VAR_GLOBAL  (* GVL_META_GOVERNANCE_FABRIC *)
  Meta_Governance_Valid : BOOL := FALSE;
  Meta_Governance_Granted : BOOL := FALSE;
  Meta_Governance_Quarantine_Active : BOOL := TRUE;
  Governance_Graph_Acyclic : BOOL := FALSE;
  Authority_Rooting_Valid : BOOL := FALSE;
  Independent_Validation_Preserved : BOOL := FALSE;
  Meta_Consistency_Coherent : BOOL := FALSE;
  Recursive_Trust_Boundaries_Stable : BOOL := FALSE;
  Validator_Independence_Valid : BOOL := FALSE;
  CrossLayer_Causality_Grounded : BOOL := FALSE;
  Bootstrap_Validation_Absent : BOOL := FALSE;
  SelfReference_Elimination_Valid : BOOL := FALSE;
  Recursive_Authority_Dependency_Detected : BOOL := FALSE;
  Circular_Validation_Chain_Detected : BOOL := FALSE;
  SelfJustifying_Governance_State_Detected : BOOL := FALSE;
  Epistemic_Recursion_Leakage_Detected : BOOL := FALSE;
  Authority_Bootstrap_Paradox_Detected : BOOL := FALSE;
  Meta_Consistency_Erosion_Detected : BOOL := FALSE;
  Meta_Governance_Epoch : UDINT := 0;
  Meta_Governance_Epoch_Coherent : BOOL := FALSE;
  Meta_Governance_Last_Update_MS : UDINT := 0;
  Meta_Governance_Lease_Expired : BOOL := TRUE;
  Meta_Governance_Last_Error_Code : UDINT := 0;
  Meta_Governance_Last_Error_Text : STRING(160) := '';
  Meta_Governance_Invalidation_Count : UDINT := 0;
END_VAR

VAR_GLOBAL  (* GVL_RECOVERY_REACTIVATION_CONTROL_FABRIC *)
  Recovery_Reactivation_Control_Valid : BOOL := FALSE;
  Recovery_Reactivation_Control_Granted : BOOL := FALSE;
  Recovery_Reactivation_Boundary_Stable : BOOL := FALSE;
  CrossSubsystem_Reactivation_Consistent : BOOL := FALSE;
  Reactivation_Energy_Boundary_Safe : BOOL := FALSE;
  Reactivation_Causality_Grounded : BOOL := FALSE;
  Reactivation_Ordering_Stable : BOOL := FALSE;
  Unsafe_Reactivation_Ordering_Detected : BOOL := FALSE;
  Partial_Reactivation_Leak_Detected : BOOL := FALSE;
  CrossSubsystem_Reactivation_Fork : BOOL := FALSE;
  Recovery_Reactivation_Epoch : UDINT := 0;
END_VAR

VAR_GLOBAL  (* GVL_GLOBAL_AUTHORITY_SYNC *)
  Global_Authority_Sync_Valid : BOOL := FALSE;
  Global_Authority_Sync_Granted : BOOL := FALSE;
  Global_Authority_Sync_Quarantine_Active : BOOL := TRUE;
  Heating_Authority_Coherent : BOOL := FALSE;
  Ventilation_Authority_Coherent : BOOL := FALSE;
  Water_Authority_Coherent : BOOL := FALSE;
  Access_Authority_Coherent : BOOL := FALSE;
  Lighting_Authority_Coherent : BOOL := FALSE;
  Cross_Domain_Epoch_Coherent : BOOL := FALSE;
  Distributed_Authority_Generation_Coherent : BOOL := FALSE;
  Global_Causality_Timeline_Stable : BOOL := FALSE;
  Multi_Domain_Recovery_Coherent : BOOL := FALSE;
  Authority_Epoch_Fragmentation_Detected : BOOL := FALSE;
  Partial_Recovery_SplitBrain_Detected : BOOL := FALSE;
  Cross_Domain_Replay_Skew_Detected : BOOL := FALSE;
  Distributed_Authority_Divergence_Detected : BOOL := FALSE;
  Global_Causality_Desynchronization_Detected : BOOL := FALSE;
  Multi_Domain_Chronology_Drift_Detected : BOOL := FALSE;
  Global_Authority_Epoch : UDINT := 0;
  Global_Authority_Epoch_Coherent : BOOL := FALSE;
  Global_Authority_Last_Update_MS : UDINT := 0;
  Global_Authority_Lease_Expired : BOOL := TRUE;
  Global_Authority_Last_Error_Code : UDINT := 0;
  Global_Authority_Last_Error_Text : STRING(160) := '';
  Global_Authority_Invalidation_Count : UDINT := 0;
END_VAR

{attribute 'qualified_only'}
VAR_GLOBAL  (* GVL_SAFETY_RECOVERY_CONFIG *)
  G_Stabilization_Delay_MS : UDINT := 5000;
  G_Stable_Time_Required_MS : UDINT := 3000;
  G_Cooldown_Time_MS : UDINT := 10000;
END_VAR

VAR_GLOBAL  (* GVL_DISTRIBUTED_FORWARD_PROGRESS_FABRIC *)
  Distributed_Forward_Progress_Valid : BOOL := FALSE;
  Distributed_Forward_Progress_Granted : BOOL := FALSE;
  Distributed_Forward_Progress_Canonical : BOOL := FALSE;
  Cluster_Progress_Consensus_Stable : BOOL := FALSE;
  Distributed_Recovery_Progress_Valid : BOOL := FALSE;
  Distributed_Progress_Causality_Valid : BOOL := FALSE;
  Cluster_Execution_Lineage_Coherent : BOOL := FALSE;
  Distributed_Livelock_Detected : BOOL := FALSE;
  Cluster_Progress_Fork_Detected : BOOL := FALSE;
  Distributed_Consensus_Progress_Deadlock : BOOL := FALSE;
  Distributed_Forward_Progress_Epoch : UDINT := 0;
END_VAR

VAR_GLOBAL  (* GVL_TELEMETRY *)
  Telemetry_Runtime_Valid : BOOL := FALSE;
  Telemetry_Freshness_Valid : BOOL := FALSE;
  Telemetry_Lease_Expired : BOOL := TRUE;
  Telemetry_Quarantine_Active : BOOL := TRUE;
  Command_Telemetry_Causality_Valid : BOOL := FALSE;
  Command_Telemetry_Divergence_Detected : BOOL := TRUE;
  Command_Epoch : UDINT := 0;
  Telemetry_Epoch : UDINT := 0;
  Last_Acknowledged_Command_Epoch : UDINT := 0;
  Actuator_Feedback_Valid : BOOL := FALSE;
  Actuator_Feedback_Fresh : BOOL := FALSE;
  Physical_Effect_Confirmed : BOOL := FALSE;
  Physical_Effect_Finalized : BOOL := FALSE;
  Physical_Target_Converged : BOOL := FALSE;
  Physical_Stable_Window_OK : BOOL := FALSE;
  Physical_Oscillation_Detected : BOOL := FALSE;
  Physical_Transition_Active : BOOL := FALSE;
  Physical_Convergence_Replay_Suspected : BOOL := FALSE;
  Telemetry_Replay_Suspected : BOOL := FALSE;
  Last_Physical_Ack_Time_MS : UDINT := 0;
  Last_Physical_Convergence_MS : UDINT := 0;
  Telemetry_Last_Error_Code : UDINT := 0;
  Telemetry_Last_Error_Text : STRING(160) := '';
  Telemetry_Invalidation_Count : UDINT := 0;
END_VAR

VAR_GLOBAL RETAIN  (* GVL_PERSISTENT *)
  P_System_Mode : E_System_Operating_Mode;
  P_Safety_Gas_Latched : BOOL;
  P_Safety_Smoke_Latched : BOOL;
  P_Safety_Leak_Latched : BOOL;
  P_DHW_Heating_Active : BOOL;
  P_Valid : BOOL;
END_VAR

VAR_GLOBAL  (* GVL_WATER_OUTPUT *)
  DO_Water_Valve_35_Close : BOOL := FALSE;
  DO_Water_Valve_36_Close : BOOL := FALSE;
  DO_Water_Zone_Enable : ARRAY[1..GVL_CONSTANTS.C_MAX_WATER_ZONES] OF BOOL;
END_VAR

VAR_GLOBAL  (* GVL_PEER_SESSION *)
  Remote_Session_Valid : BOOL := FALSE;
  Remote_Last_Refresh_MS : UDINT := 0;
  Remote_Runtime_Epoch : ULINT := 0;
  Remote_Snapshot_Epoch : ULINT := 0;
  Remote_Boot_Generation : ULINT := 0;
  Remote_Fencing_Token : ULINT := 0;
  Remote_Publication_Allowed : BOOL := FALSE;
  Remote_Runtime_Healthy : BOOL := FALSE;
END_VAR

{attribute 'qualified_only'}
VAR_GLOBAL  (* GVL_TEST_PANEL *)
  G_Enable : BOOL := FALSE;
  G_Scenario_ID : INT := 1;
  G_Scenario_ID_Prev : INT := 0;
  G_Scenario_Run : BOOL := FALSE;
  G_Scenario_Active : BOOL := FALSE;
  G_UI_00_Header : STRING(200) := '=== TEST PANEL ===';
  G_UI_01_Test : STRING(200) := 'Select G_Scenario_ID';
  G_UI_02_Change : STRING(200) := 'CHANGE: set scenario inputs';
  G_UI_03_Expected : STRING(200) := 'EXPECTED: see scenario instruction';
  G_UI_04_Result : STRING(200) := 'RESULT: Idle';
  G_UI_05_Error : STRING(200) := 'ERROR: -';
  G_UI_06_Actual : STRING(200) := 'ACTUAL: see numeric fields below';
  G_UI_07_Separator : STRING(200) := '----------------------------------------';
  G_UI_10_Numeric_Block : STRING(200) := 'NUMERIC: Base / Expected / Actual / Delta';
  G_UI_11_Array_Block : STRING(200) := 'ARRAYS: Manifold expected / actual / enabled';
  G_UI_12_State_Block : STRING(200) := 'STATE: Safety / Block / Budget / Preheat';
  G_Run_Counter : UDINT := 0;
  G_Last_Scenario_ID : INT := 0;
  G_Last_Result_Passed : BOOL := TRUE;
  G_Last_Fail_Code : UDINT := 0;
  G_Reset_Results_Request : BOOL := FALSE;
  G_Reset_Inputs_Request : BOOL := FALSE;
  G_Current_Test_Name : STRING(200) := '';
  G_Expected_Summary : STRING(200) := '';
  G_Actual_Summary : STRING(200) := '';
  G_Test_Result_Line : STRING(200) := 'Idle';
  G_Last_Result_Line : STRING(200) := '';
  G_Error_Text : STRING(200) := '';
  G_System_State_Line : STRING(200) := '';
  G_Selected_Circuit : INT := 1;
  G_Input_Policy_Bias : INT := 0;
  G_Input_Guest_Preheat_Request : BOOL := FALSE;
  G_Input_Guest_Preheat_Enabled : BOOL := TRUE;
  G_Input_Guest_Preheat_Boost : INT := 2;
  G_Input_Max_Thermal_Budget : REAL := 2.0;
  G_Input_Block_Heating : BOOL := FALSE;
  G_Input_Safety_Stop : BOOL := FALSE;
  G_Input_Circuit_Enable : ARRAY[1..GVL_CONSTANTS.C_MAX_HEATING_CIRCUITS] OF BOOL;
  G_Input_Circuit_Bias : ARRAY[1..GVL_CONSTANTS.C_MAX_HEATING_CIRCUITS] OF INT;
  G_Input_Circuit_Guest_Preheat : ARRAY[1..GVL_CONSTANTS.C_MAX_HEATING_CIRCUITS] OF BOOL;
  G_Test_Description : STRING(200) := 'Idle';
  G_Test_What_To_Change : STRING(200) := '';
  G_Test_Expected_Text : STRING(200) := '';
  G_Result_Mapped_Manifold : INT := 0;
  G_Result_Base_Priority : INT := 0;
  G_Result_Expected_Adjusted_Priority : INT := 0;
  G_Result_Actual_Adjusted_Priority : INT := 0;
  G_Result_Delta : INT := 0;
  G_Result_Manifold_Base_Priority : ARRAY[1..GVL_CONSTANTS.C_MAX_MANIFOLDS] OF INT;
  G_Result_Manifold_Expected_Priority : ARRAY[1..GVL_CONSTANTS.C_MAX_MANIFOLDS] OF INT;
  G_Result_Manifold_Actual_Priority : ARRAY[1..GVL_CONSTANTS.C_MAX_MANIFOLDS] OF INT;
  G_Result_Manifold_Delta : ARRAY[1..GVL_CONSTANTS.C_MAX_MANIFOLDS] OF INT;
  G_Result_Manifold_Allowed : ARRAY[1..GVL_CONSTANTS.C_MAX_MANIFOLDS] OF BOOL;
  G_Result_Manifold_Enabled : ARRAY[1..GVL_CONSTANTS.C_MAX_MANIFOLDS] OF BOOL;
  G_Result_Used_Thermal_Budget : REAL := 0.0;
  G_Result_Budget_Exceeded : BOOL := FALSE;
  G_Result_Passed : BOOL := TRUE;
  G_Result_Status_Msg : STRING(200) := 'Idle';
  G_Result_Fail_Code : UDINT := 0;
END_VAR

VAR_GLOBAL  (* GVL_LIGHTING_OUTPUT *)
  AO_Lighting_Levels : ARRAY[1..GVL_CONSTANTS.C_MAX_LIGHT_ZONES] OF UINT;
  AO_Blinds_Positions : ARRAY[1..GVL_CONSTANTS.C_MAX_BLINDS] OF UINT;
  DO_Sockets : ARRAY[1..GVL_CONSTANTS.C_MAX_SOCKETS] OF BOOL;
END_VAR

VAR_GLOBAL  (* GVL_DETERMINISTIC_RECOVERY_PATH_FABRIC *)
  Deterministic_Recovery_Path_Valid : BOOL := FALSE;
  Deterministic_Recovery_Path_Granted : BOOL := FALSE;
  Deterministic_Recovery_Path_Quarantine_Active : BOOL := TRUE;
  Deterministic_Recovery_Path_Canonical : BOOL := FALSE;
  Recovery_Lineage_Causality_Valid : BOOL := FALSE;
  Recovery_Physical_Convergence_Stable : BOOL := FALSE;
  Recovery_Timeline_Monotonic : BOOL := FALSE;
  Recovery_Causality_Grounded : BOOL := FALSE;
  Recovery_Path_Continuity_Valid : BOOL := FALSE;
  Distributed_Recovery_Consensus_Valid : BOOL := FALSE;
  Unsafe_Recovery_Path_Detected : BOOL := FALSE;
  Recovery_Path_Divergence_Detected : BOOL := FALSE;
  Recovery_Causality_Break_Detected : BOOL := FALSE;
  Distributed_Recovery_Fork_Detected : BOOL := FALSE;
  Deterministic_Recovery_Path_Epoch : UDINT := 0;
  Deterministic_Recovery_Path_Last_Update_MS : UDINT := 0;
END_VAR

VAR_GLOBAL  (* GVL_ENERGY_CAUSALITY_FABRIC *)
  Energy_Causality_Valid : BOOL := FALSE;
  Energy_Causality_Granted : BOOL := FALSE;
  Energy_Causality_Quarantine_Active : BOOL := TRUE;
  Hydraulic_Energy_State_Valid : BOOL := FALSE;
  Thermal_Energy_State_Valid : BOOL := FALSE;
  Electrical_Load_State_Valid : BOOL := FALSE;
  Motor_Energy_Envelope_Valid : BOOL := FALSE;
  Distributed_Load_Coherent : BOOL := FALSE;
  Energy_Envelope_Stable : BOOL := FALSE;
  Transient_Load_Stable : BOOL := FALSE;
  Thermal_Accumulation_Stable : BOOL := FALSE;
  Recovery_Energy_Coherent : BOOL := FALSE;
  DryRun_Energy_State_Detected : BOOL := FALSE;
  Thermal_Extraction_Divergence_Detected : BOOL := FALSE;
  Load_Synchronization_Spike_Detected : BOOL := FALSE;
  Hydraulic_Energy_Starvation_Detected : BOOL := FALSE;
  Distributed_Transient_Overload_Detected : BOOL := FALSE;
  Energy_Recovery_Instability_Detected : BOOL := FALSE;
  Energy_Causality_Epoch : UDINT := 0;
  Energy_Causality_Epoch_Coherent : BOOL := FALSE;
  Energy_Causality_Last_Update_MS : UDINT := 0;
  Energy_Causality_Lease_Expired : BOOL := TRUE;
  Energy_Causality_Last_Error_Code : UDINT := 0;
  Energy_Causality_Last_Error_Text : STRING(160) := '';
  Energy_Causality_Invalidation_Count : UDINT := 0;
END_VAR

{attribute 'qualified_only'}
VAR_GLOBAL  (* GVL_MODBUS_SYSCOM_TRANSPORT *)
  G_Transport_Enabled : BOOL := FALSE;
  G_Transport_Attached : BOOL := FALSE;
  G_Backend_State : E_Modbus_SysCom_Backend_State := MB_SYSCOM_CLOSED;
  G_Backend_Last_Error_MS : UDINT := 0;
  G_Backend_Reconnect_Delay_MS : UDINT := 3000;
  G_Backend_Reconnect_Attempts : UDINT := 0;
  G_Backend_Online : BOOL := FALSE;
  G_TX_Request : BOOL := FALSE;
  G_TX_Buffer : ARRAY[0..255] OF BYTE;
  G_TX_Length : UINT := 0;
  G_TX_Done : BOOL := FALSE;
  G_TX_Error : BOOL := FALSE;
  G_TX_Error_Code : WORD := 0;
  G_RX_Ready : BOOL := FALSE;
  G_RX_Buffer : ARRAY[0..255] OF BYTE;
  G_RX_Length : UINT := 0;
  G_RX_Error : BOOL := FALSE;
  G_RX_Error_Code : WORD := 0;
  G_RX_State : E_Modbus_RTU_RX_State := MB_RTU_RX_IDLE;
  G_RX_Assembler_Active : BOOL := FALSE;
  G_RX_Assembler_Length : UINT := 0;
  G_RX_Assembler_Last_Byte_MS : UDINT := 0;
  G_RX_Assembler_InterFrame_MS : UDINT := 20;
  G_RX_Assembler_Overflow : BOOL := FALSE;
  G_RX_Assembler_CRC_OK : BOOL := FALSE;
  G_RX_Assembler_CRC_Frame : WORD := 0;
  G_RX_Assembler_CRC_Calc : WORD := 0;
  G_Last_TX_Request_MS : UDINT := 0;
  G_Last_TX_Done_MS : UDINT := 0;
  G_Last_RX_MS : UDINT := 0;
  G_TX_Watchdog_Timeout : BOOL := FALSE;
  G_RX_Watchdog_Timeout : BOOL := FALSE;
  G_Bus_Silent : BOOL := FALSE;
  G_Total_TX : UDINT := 0;
  G_Total_RX : UDINT := 0;
  G_Total_Errors : UDINT := 0;
  G_Total_RX_Overflow : UDINT := 0;
  G_Total_RX_Short_Frame : UDINT := 0;
  G_Total_RX_CRC_Error : UDINT := 0;
  G_Total_Reconnects : UDINT := 0;
  G_Total_TX_Watchdog : UDINT := 0;
  G_Total_RX_Watchdog : UDINT := 0;
END_VAR

VAR_GLOBAL  (* GVL_PLC_FENCING *)
  PLC_Ownership_Epoch : ULINT := 0;
  PLC_Fencing_Token : ULINT := 0;
  PLC_Ownership_Valid : BOOL := FALSE;
  PLC_Semantic_Authority_Valid : BOOL := FALSE;
  PLC_Heartbeat_Only_Mode : BOOL := FALSE;
  PLC_Lease_Active : BOOL := FALSE;
  PLC_Lease_Expired : BOOL := FALSE;
  PLC_Lease_Timeout_MS : UDINT := 5000;
  PLC_Last_Lease_Refresh_MS : UDINT := 0;
  PLC_Last_Authority_Validation_MS : UDINT := 0;
  PLC_Split_Brain_Detected : BOOL := FALSE;
  PLC_Stale_Owner_Detected : BOOL := FALSE;
  PLC_Asymmetric_Partition_Detected : BOOL := FALSE;
  PLC_Forced_Safe_Quarantine : BOOL := FALSE;
  PLC_Last_Error_Code : UDINT := 0;
  PLC_Last_Error_Text : STRING(160) := '';
  PLC_Fencing_Invalidation_Count : UDINT := 0;
END_VAR

VAR_GLOBAL  (* GVL_AUTHORITY_REVOCATION *)
  Authority_Revocation_Active : BOOL := FALSE;
  Authority_Revocation_Propagated : BOOL := FALSE;
  Authority_Fail_Closed_Valid : BOOL := FALSE;
  Snapshot_Authority_Revoked : BOOL := FALSE;
  Sensor_Consensus_Authority_Revoked : BOOL := FALSE;
  Telemetry_Causality_Authority_Revoked : BOOL := FALSE;
  Physical_Authority_Epoch_Revoked : BOOL := FALSE;
  Authority_Lineage_Revoked : BOOL := FALSE;
  PreOutput_Authority_Revoked : BOOL := FALSE;
  Physical_IO_Release_Denied : BOOL := FALSE;
  Quarantine_Fabric_Active : BOOL := FALSE;
  Revocation_Order_Valid : BOOL := FALSE;
  Revocation_Replay_Suspected : BOOL := FALSE;
  Partial_Revocation_Detected : BOOL := FALSE;
  Stale_Downstream_Authority_Detected : BOOL := FALSE;
  Revocation_Epoch : UDINT := 0;
  Revocation_Last_Update_MS : UDINT := 0;
  Revocation_Last_Error_Code : UDINT := 0;
  Revocation_Last_Error_Text : STRING(160) := '';
  Revocation_Invalidation_Count : UDINT := 0;
END_VAR

VAR_GLOBAL  (* GVL_PROVENANCE_CONTINUITY_FABRIC *)
  Provenance_Continuity_Valid : BOOL := FALSE;
  Provenance_Continuity_Granted : BOOL := FALSE;
  Provenance_Continuity_Quarantine_Active : BOOL := TRUE;
  Recovery_Provenance_Reattested : BOOL := FALSE;
  Authority_Resurrection_Authentic : BOOL := FALSE;
  Federation_Rejoin_Provenance_Valid : BOOL := FALSE;
  PostRecovery_TrustSeed_Coherent : BOOL := FALSE;
  CrossEpoch_Provenance_Continuity_Stable : BOOL := FALSE;
  Recovery_Epoch_Authenticity_Valid : BOOL := FALSE;
  Distributed_Rejoin_Attestation_Coherent : BOOL := FALSE;
  Authority_Restoration_Provenance_Grounded : BOOL := FALSE;
  Provenance_Lease_Continuity_Valid : BOOL := FALSE;
  Stale_Provenance_Resurrection_Detected : BOOL := FALSE;
  Recovered_Authority_Without_Reattestation_Detected : BOOL := FALSE;
  Federation_Rejoin_Without_Provenance_Detected : BOOL := FALSE;
  CrossEpoch_Trust_Continuity_Broken : BOOL := FALSE;
  Recovery_Trust_Seed_Drift_Detected : BOOL := FALSE;
  Provenance_Resurrection_Bypass_Detected : BOOL := FALSE;
  Provenance_Continuity_Epoch : UDINT := 0;
  Provenance_Continuity_Epoch_Coherent : BOOL := FALSE;
  Provenance_Continuity_Last_Update_MS : UDINT := 0;
  Provenance_Continuity_Lease_Expired : BOOL := TRUE;
  Provenance_Continuity_Last_Error_Code : UDINT := 0;
  Provenance_Continuity_Last_Error_Text : STRING(160) := '';
  Provenance_Continuity_Invalidation_Count : UDINT := 0;
END_VAR

{attribute 'qualified_only'}
VAR_GLOBAL  (* GVL_COMMAND *)
  G_Gas_Valve_Close : BOOL := FALSE;
  G_Boiler_Stop : BOOL := FALSE;
  G_Supply_100_Req : BOOL := FALSE;
  G_Supply_80_Req : BOOL := FALSE;
  G_Vent_PV3_Boost : BOOL := FALSE;
  G_Exhaust_100_Req : BOOL := FALSE;
  G_Vent_Stop : BOOL := FALSE;
  G_Close_Valve_35 : BOOL := FALSE;
  G_Close_Valve_36 : BOOL := FALSE;
  G_Gate_Open : BOOL;
  G_Wicket_Open : BOOL;
  G_Lock_1_Open : BOOL;
  G_Lock_1_Close : BOOL;
  G_Lock_2_Open : BOOL;
  G_Lock_2_Close : BOOL;
  G_Reset_Errors : BOOL := FALSE;
  G_Scenario_Request : E_SCENARIO_TYPE := E_SCENARIO_TYPE.SCENARIO_NONE;
  G_Scenario_Request_Operator : E_SCENARIO_TYPE := E_SCENARIO_TYPE.SCENARIO_NONE;
  G_Arm_Req : BOOL;
  G_Disarm_Req : BOOL;
  G_PIN_Code : STRING(4);
  G_RFID_Tag : STRING(20);
  G_2FA_Code_In : STRING(6);
  G_Send_2FA_Req : BOOL;
  G_2FA_Code_Out : STRING(6);
  G_Lighting_Override : ARRAY[1..GVL_CONSTANTS.C_MAX_LIGHT_ZONES] OF BYTE;
  G_Blinds_Override : ARRAY[1..GVL_CONSTANTS.C_MAX_BLINDS] OF BYTE;
  G_Socket_Override : ARRAY[1..GVL_CONSTANTS.C_MAX_SOCKETS] OF BOOL;
  CMD_Set_Manifold_Pump_In_Service : ARRAY[1..GVL_CONSTANTS.C_MAX_MANIFOLDS] OF BOOL;
  CMD_Set_DHW_Heating_Pump_In_Service : BOOL;
  CMD_Set_DHW_Circ_Pump_In_Service : BOOL;
  CMD_Dangerous_Action_Confirm : BOOL;
  CMD_Dangerous_Action_Request : BOOL;
  CMD_User_Access_Level : INT := 0;
  CMD_Valve_Test_Open : BOOL;
  CMD_Valve_Test_Close : BOOL;
  CMD_Valve_Test_Confirm : BOOL;
  CMD_Water_Valve_Test_Open : BOOL;
  CMD_Water_Valve_Test_Close : BOOL;
  CMD_Water_Valve_Test_Confirm : BOOL;
  CMD_Gas_Valve_Test_Open : BOOL;
  CMD_Gas_Valve_Test_Close : BOOL;
  CMD_Gas_Valve_Test_Confirm : BOOL;
  CMD_Water_Selective_Recover : BOOL;
  CMD_Gas_Selective_Recover : BOOL;
END_VAR

{attribute 'qualified_only'}
VAR_GLOBAL  (* GVL_TEST_PANEL_RESULT *)
  G_Enable : BOOL := FALSE;
  G_Scenario_ID : INT := 0;
  G_Scenario_Run : BOOL := FALSE;
  G_Scenario_Active : BOOL := FALSE;
  G_Test_Result_Line : STRING(200) := 'Idle';
  G_Result_Passed : BOOL := FALSE;
  G_Result_Status_Msg : STRING(200) := 'Idle';
  G_Result_Fail_Code : UDINT := 0;
  G_Result_Base_Priority : INT := 0;
  G_Result_Expected_Adjusted_Priority : INT := 0;
  G_Result_Actual_Adjusted_Priority : INT := 0;
  G_Result_Delta : INT := 0;
  G_Result_Budget_Exceeded : BOOL := FALSE;
  G_Result_Used_Thermal_Budget : REAL := 0.0;
  G_Result_Manifold_Enabled : ARRAY[1..GVL_CONSTANTS.C_MAX_MANIFOLDS] OF BOOL;
END_VAR

{attribute 'qualified_only'}
VAR_GLOBAL  (* GVL_Water_Isolation_Authority *)
  G_Authority_State : ARRAY[1..GVL_CONSTANTS.C_MAX_FLOOD_SENSORS] OF ST_Water_Isolation_Authority_State;
  G_Any_Selective_Authority_Allowed : BOOL;
  G_Any_Global_Fallback_Required : BOOL;
  G_Any_Authority_Denied : BOOL;
  G_Authority_Valid : BOOL;
  G_Last_Update_MS : UDINT;
  G_Status_Code : UINT;
  G_Status_Text : STRING(128);
END_VAR

{attribute 'qualified_only'}
VAR_GLOBAL  (* GVL_HEATING_POLICY_CONFIG *)
  G_Guest_Preheat_Enabled : BOOL := TRUE;
  G_Guest_Preheat_Priority_Boost : INT := 2;
  G_Guest_Preheat_Max_Duration_MS : UDINT := 7200000;
  G_Zone_Schedule : ARRAY[1..GVL_CONSTANTS.C_MAX_ZONES, 1..3] OF ST_Heating_Schedule_Event;
END_VAR

{attribute 'qualified_only'}
VAR_GLOBAL  (* GVL_Water_Topology_Validation *)
  G_Validation_State : ARRAY[1..64] OF ST_Water_Topology_Validation_State;
  G_Any_Invalid : BOOL;
  G_Any_Ambiguous : BOOL;
  G_Any_Global_Fallback_Required : BOOL;
  G_Runtime_Valid : BOOL;
  G_Last_Update_MS : UDINT;
  G_Status_Code : UINT;
  G_Status_Text : STRING(128);
END_VAR

{attribute 'qualified_only'}
VAR_GLOBAL  (* GVL_TIME_SERVICE *)
  G_Now_MS : UDINT;
  G_Time_Of_Day_MS : UDINT;
  G_Current_TOD : TOD;
  G_Day_Of_Week : INT;
  G_Last_Now_MS : UDINT;
  G_Delta_MS : UDINT;
  G_Wrap_Detected : BOOL;
  G_Sim_Enabled : BOOL;
  G_Sim_Frozen : BOOL;
  G_Sim_Time_Scale : REAL := 1.0;
  G_Sim_Now_MS : UDINT;
  G_Sim_Time_Of_Day_MS : UDINT;
  G_Sim_Day_Of_Week : INT := 1;
END_VAR

VAR_GLOBAL  (* GVL_INTENT_SYSTEM *)
  I_Source_Valid : BOOL := FALSE;
  I_Last_Update_Cycle : UDINT := 0;
  I_Last_Update_MS : UDINT := 0;
  I_Mode_Safe_Stop_Active : BOOL := FALSE;
  I_Mode_Degraded_Active : BOOL := FALSE;
  I_Mode_Freeze_Protection_Active : BOOL := FALSE;
  I_Preheat_Request : BOOL := FALSE;
  I_Freeze_Request : BOOL := FALSE;
  I_Scenario_Request_Allowed : BOOL := FALSE;
  I_Operator_Scenario_Block : BOOL := FALSE;
  I_Gateway_Command_Valid : BOOL := FALSE;
  I_Gateway_Command_Type : INT := 0;
  I_Gateway_Writes_Allowed : BOOL := FALSE;
  I_Reset_Errors_Request : BOOL := FALSE;
  I_Config_Apply_Allowed : BOOL := FALSE;
  I_Time_Sync_Allowed : BOOL := FALSE;
  I_Temperature_Write_Allowed : BOOL := FALSE;
  I_Ventilation_Write_Allowed : BOOL := FALSE;
  I_Maintenance_Apply_Allowed : BOOL := FALSE;
  I_Lighting_Overrides_Block : BOOL := FALSE;
  I_Blinds_Overrides_Block : BOOL := FALSE;
  I_Socket_Overrides_Block : BOOL := FALSE;
  I_Access_Open_Allowed : BOOL := FALSE;
  I_Manual_Override_Allowed : BOOL := FALSE;
  I_Dangerous_Action_Allowed : BOOL := FALSE;
END_VAR

VAR_GLOBAL  (* GVL_EVENT *)
  G_Event_Log : ARRAY[0..63] OF ST_EVENT;
  G_Event_Head : UINT;
  G_Event_ID_Counter : UDINT;
END_VAR

{attribute 'qualified_only'}
VAR_GLOBAL  (* GVL_Heating_Source_Stability *)
  G_State : ARRAY[1..GVL_CONSTANTS.C_MAX_HEATING_CIRCUITS] OF ST_Heating_Runtime_Source_Instability_State;
END_VAR

VAR_GLOBAL  (* GVL_PHYSICAL_TRANSACTION *)
  Physical_Transaction_Valid : BOOL := FALSE;
  Physical_Transaction_Granted : BOOL := FALSE;
  Physical_Transaction_Quarantine_Active : BOOL := TRUE;
  Physical_Transaction_Epoch : UDINT := 0;
  Physical_Transaction_Command_Epoch : UDINT := 0;
  Physical_Transaction_ACK_Epoch : UDINT := 0;
  All_Actuators_Converged : BOOL := FALSE;
  Cross_Actuator_Epoch_Coherent : BOOL := FALSE;
  Distributed_Actuation_Coherent : BOOL := FALSE;
  Stable_Plant_State_Confirmed : BOOL := FALSE;
  Valve_Transition_Confirmed : BOOL := FALSE;
  Pump_Transition_Confirmed : BOOL := FALSE;
  Damper_Transition_Confirmed : BOOL := FALSE;
  Relay_Bank_Transition_Confirmed : BOOL := FALSE;
  Flow_Stabilization_Confirmed : BOOL := FALSE;
  Pressure_Stabilization_Confirmed : BOOL := FALSE;
  Thermal_Response_Confirmed : BOOL := FALSE;
  Electrical_Load_Stabilized : BOOL := FALSE;
  Partial_Plant_Transition_Detected : BOOL := FALSE;
  Cross_Actuator_Convergence_Skew : BOOL := FALSE;
  Pump_Valve_Ordering_Race_Detected : BOOL := FALSE;
  Distributed_Actuator_Rollback_Detected : BOOL := FALSE;
  Transaction_Timeout_Detected : BOOL := FALSE;
  Brownout_Partial_Switching_Detected : BOOL := FALSE;
  Physical_Transaction_Last_Update_MS : UDINT := 0;
  Physical_Transaction_Lease_Expired : BOOL := TRUE;
  Physical_Transaction_Last_Error_Code : UDINT := 0;
  Physical_Transaction_Last_Error_Text : STRING(160) := '';
  Physical_Transaction_Invalidation_Count : UDINT := 0;
END_VAR

{attribute 'qualified_only'}
VAR_GLOBAL  (* GVL_Water_Isolation_Intent *)
  G_Zone_Close_Requested : ARRAY[1..GVL_CONSTANTS.C_MAX_FLOOD_SENSORS] OF BOOL;
  G_Valve_Group_Close_Requested : ARRAY[1..GVL_CONSTANTS.C_MAX_FLOOD_SENSORS] OF BOOL;
  G_Global_Isolation_Requested : BOOL;
  G_Intent_Valid : BOOL;
  G_Status_Code : UINT;
  G_Status_Text : STRING(128);
END_VAR

VAR_GLOBAL  (* GVL_TEMPORAL_STABILITY *)
  Temporal_Stability_Valid : BOOL := FALSE;
  Temporal_Stability_Granted : BOOL := FALSE;
  Temporal_Stability_Quarantine_Active : BOOL := TRUE;
  Stability_Observation_Window_Active : BOOL := FALSE;
  Stability_Window_Start_MS : UDINT := 0;
  Stability_Window_Elapsed_MS : UDINT := 0;
  Stability_Window_Target_MS : UDINT := 5000;
  Post_Convergence_Stable : BOOL := FALSE;
  No_Oscillation_Detected : BOOL := FALSE;
  No_Relay_Chatter_Detected : BOOL := FALSE;
  Thermal_Slope_Stable : BOOL := FALSE;
  Pressure_Stable : BOOL := FALSE;
  Flow_Stable : BOOL := FALSE;
  Post_Convergence_Oscillation_Detected : BOOL := FALSE;
  Thermal_Inertia_Rebound_Detected : BOOL := FALSE;
  Pressure_Rebound_Detected : BOOL := FALSE;
  Relay_Chatter_Detected : BOOL := FALSE;
  Pump_Cavitation_Recovery_Detected : BOOL := FALSE;
  Delayed_Actuator_Divergence_Detected : BOOL := FALSE;
  Temporal_Stability_Epoch : UDINT := 0;
  Temporal_Stability_Epoch_Coherent : BOOL := FALSE;
  Temporal_Stability_Last_Update_MS : UDINT := 0;
  Temporal_Stability_Lease_Expired : BOOL := TRUE;
  Temporal_Stability_Last_Error_Code : UDINT := 0;
  Temporal_Stability_Last_Error_Text : STRING(160) := '';
  Temporal_Stability_Invalidation_Count : UDINT := 0;
END_VAR

{attribute 'qualified_only'}
VAR_GLOBAL  (* GVL_Water_Output_Projection *)
  G_Output_Projection_State : ARRAY[1..64] OF ST_Water_Output_Projection_State;
  G_Any_Output_Projected : BOOL;
  G_Any_Projection_Denied : BOOL;
  G_Global_Fallback_Projecting : BOOL;
  G_Runtime_Valid : BOOL;
  G_Last_Update_MS : UDINT;
  G_Status_Code : UINT;
  G_Status_Text : STRING(128);
END_VAR

VAR_GLOBAL  (* GVL_OPERATIONAL_INTELLIGENCE_FABRIC *)
  Operational_Intelligence_Active : BOOL := TRUE;
  Operational_Intelligence_ReadOnly : BOOL := TRUE;
  Operational_Intelligence_NoMutation : BOOL := TRUE;
  Dominant_Instability_Source_Available : BOOL := FALSE;
  Active_Degradation_Cause_Available : BOOL := FALSE;
  Recovery_Blocker_Observed : BOOL := FALSE;
  Governance_Pressure_Hotspot_Observed : BOOL := FALSE;
  Operational_Reasoning_Consistency_Valid : BOOL := FALSE;
  Runtime_Causal_Projection_Valid : BOOL := FALSE;
  Distributed_Operational_Context_Valid : BOOL := FALSE;
  Governance_Saturation_Observed : BOOL := FALSE;
  Governance_Complexity_Pressure_Observed : BOOL := FALSE;
  Operational_Opacity_Observed : BOOL := FALSE;
  Operational_Intelligence_Epoch : UDINT := 0;
END_VAR

{attribute 'qualified_only'}
VAR_GLOBAL  (* GVL_DIAGNOSTICS_EXT *)
  G_Health_Heating : REAL := 1.0;
  G_Health_Safety : REAL := 1.0;
  G_Health_IO : REAL := 1.0;
  G_Error_Count_Heating : UDINT := 0;
  G_Error_Count_Safety : UDINT := 0;
  G_Error_Count_IO : UDINT := 0;
  G_Last_Error_Time_Heating : UDINT := 0;
  G_Last_Error_Time_Safety : UDINT := 0;
  G_Last_Error_Time_IO : UDINT := 0;
  G_Last_Update_Time : UDINT := 0;
  G_Cycle_Expected_MS : UDINT := 250;
  G_Cycle_Warning_MS : UDINT := 375;
  G_Cycle_Critical_MS : UDINT := 500;
  G_Cycle_Last_MS : UDINT := 0;
  G_Cycle_Max_MS : UDINT := 0;
  G_Cycle_Min_MS : UDINT := 0;
  G_Cycle_Avg_MS : REAL := 0.0;
  G_Cycle_Sample_Count : UDINT := 0;
  G_Cycle_Overrun_Count : UDINT := 0;
  G_Cycle_Critical_Count : UDINT := 0;
  G_Cycle_Last_Overrun_MS : UDINT := 0;
  G_Cycle_Last_Overrun_Time_MS : UDINT := 0;
  G_Cycle_Overrun_Active : BOOL := FALSE;
  G_Cycle_Critical_Active : BOOL := FALSE;
  G_Heating_State : INT := 0;  (* 0=OK,1=DEGRADED,2=CRITICAL *)
  G_Safety_State : INT := 0;
  G_IO_State : INT := 0;
END_VAR

VAR_GLOBAL  (* GVL_SAFETY_SHUTDOWN *)
  G_Safety_Mode : E_Safety_Mode := NORMAL;
  G_Safety_Active : BOOL := FALSE;
END_VAR

VAR_GLOBAL RETAIN  (* GVL_AUTHORITY_LINEAGE *)
  Authority_Lineage_Epoch : UDINT := 0;
  Authority_Lineage_Valid : BOOL := FALSE;
  Warm_Restart_Continuity_Valid : BOOL := FALSE;
  HA_Resume_Continuity_Valid : BOOL := FALSE;
  Retained_State_Integrity_Valid : BOOL := FALSE;
  Authority_Replay_Suspected : BOOL := FALSE;
  Retained_State_Skew_Detected : BOOL := FALSE;
  Partial_Authority_Resurrection_Detected : BOOL := FALSE;
  Epoch_Lineage_Discontinuity_Detected : BOOL := FALSE;
  Last_Physical_Authority_Epoch : UDINT := 0;
  Last_Runtime_Epoch : UDINT := 0;
  Last_Output_Publication_Epoch : UDINT := 0;
  Authority_Lineage_Boot_ID : UDINT := 0;
  Authority_Lineage_Last_Update_MS : UDINT := 0;
  Authority_Lineage_Last_Error_Code : UDINT := 0;
  Authority_Lineage_Last_Error_Text : STRING(160) := '';
  Authority_Lineage_Invalidation_Count : UDINT := 0;
END_VAR

VAR_GLOBAL  (* GVL_CONTROL_TIMING_FABRIC *)
  Control_Temporal_Coherence_Valid : BOOL := FALSE;
  Control_Temporal_Coherence_Granted : BOOL := FALSE;
  Control_Temporal_Coherence_Quarantine_Active : BOOL := TRUE;
  Loop_Sampling_Coherent : BOOL := FALSE;
  Feedback_Freshness_Valid : BOOL := FALSE;
  PID_Phase_Alignment_Valid : BOOL := FALSE;
  Cross_Loop_Temporal_Stable : BOOL := FALSE;
  Multi_Rate_Causality_Coherent : BOOL := FALSE;
  Control_Snapshot_Epoch_Coherent : BOOL := FALSE;
  Feedback_Window_Stable : BOOL := FALSE;
  Loop_Execution_Phase_Stable : BOOL := FALSE;
  Temporal_Observation_Aligned : BOOL := FALSE;
  PID_Phase_Skew_Detected : BOOL := FALSE;
  Sampling_Window_Divergence_Detected : BOOL := FALSE;
  Feedback_Freshness_Aliasing_Detected : BOOL := FALSE;
  Cross_Loop_Stabilization_Lag_Detected : BOOL := FALSE;
  Multi_Rate_Oscillation_Risk_Detected : BOOL := FALSE;
  Distributed_Control_Ringing_Detected : BOOL := FALSE;
  Control_Timing_Epoch : UDINT := 0;
  Control_Timing_Epoch_Coherent : BOOL := FALSE;
  Control_Timing_Last_Update_MS : UDINT := 0;
  Control_Timing_Lease_Expired : BOOL := TRUE;
  Control_Timing_Last_Error_Code : UDINT := 0;
  Control_Timing_Last_Error_Text : STRING(160) := '';
  Control_Timing_Invalidation_Count : UDINT := 0;
END_VAR

VAR_GLOBAL  (* GVL_SEMANTIC_CONTINUITY *)
  Semantic_Continuity_Valid : BOOL := FALSE;
  Semantic_Continuity_Granted : BOOL := FALSE;
  Semantic_Continuity_Quarantine_Active : BOOL := TRUE;
  Operator_Intent_Coherent : BOOL := FALSE;
  Policy_Intent_Coherent : BOOL := FALSE;
  Adaptive_Behavior_Coherent : BOOL := FALSE;
  Recovery_Intent_Coherent : BOOL := FALSE;
  Distributed_Semantic_Coherent : BOOL := FALSE;
  Declared_System_Intent_Valid : BOOL := FALSE;
  Runtime_Goal_Alignment_Valid : BOOL := FALSE;
  Optimization_Boundary_Valid : BOOL := FALSE;
  Autonomous_Adjustment_Valid : BOOL := FALSE;
  Goal_Drift_Detected : BOOL := FALSE;
  Policy_Divergence_Detected : BOOL := FALSE;
  Adaptive_Learning_Semantic_Skew : BOOL := FALSE;
  Recovery_Intent_Mismatch_Detected : BOOL := FALSE;
  Optimization_Authority_Corruption_Detected : BOOL := FALSE;
  Distributed_Semantic_Fragmentation_Detected : BOOL := FALSE;
  Semantic_Continuity_Epoch : UDINT := 0;
  Semantic_Continuity_Epoch_Coherent : BOOL := FALSE;
  Semantic_Last_Update_MS : UDINT := 0;
  Semantic_Lease_Expired : BOOL := TRUE;
  Semantic_Last_Error_Code : UDINT := 0;
  Semantic_Last_Error_Text : STRING(160) := '';
  Semantic_Invalidation_Count : UDINT := 0;
END_VAR

VAR_GLOBAL  (* GVL_CAUSAL_NARRATIVE_FABRIC *)
  Causal_Narrative_Active : BOOL := TRUE;
  Causal_Narrative_ReadOnly : BOOL := TRUE;
  Runtime_Narrative_Available : BOOL := FALSE;
  Recovery_Narrative_Available : BOOL := FALSE;
  Authority_Narrative_Available : BOOL := FALSE;
  Temporal_Narrative_Available : BOOL := FALSE;
  Narrative_Causality_Coherent : BOOL := FALSE;
  Narrative_Runtime_Alignment_Valid : BOOL := FALSE;
  Narrative_Opacity_Observed : BOOL := FALSE;
  Narrative_Gap_Observed : BOOL := FALSE;
  Runtime_Narrative_Code : STRING(255) := '';
  Recovery_Narrative_Code : STRING(255) := '';
  Authority_Narrative_Code : STRING(255) := '';
  Causal_Narrative_Epoch : UDINT := 0;
END_VAR

VAR_GLOBAL  (* GVL_DISTRIBUTED_SAFETY_REALITY_CONSENSUS_FABRIC *)
  Distributed_Safety_Reality_Consensus_Valid : BOOL := FALSE;
  Distributed_Safety_Reality_Consensus_Granted : BOOL := FALSE;
  Distributed_Safety_Consensus_Valid : BOOL := FALSE;
  Cluster_Safety_Reality_Stable : BOOL := FALSE;
  Distributed_Observability_Reality_Equivalence : BOOL := FALSE;
  Distributed_Safety_Causality_Valid : BOOL := FALSE;
  Cluster_Safety_Lineage_Coherent : BOOL := FALSE;
  Distributed_Safety_State_Fork : BOOL := FALSE;
  Cluster_Safety_Projection_Drift : BOOL := FALSE;
  Distributed_Unsafe_State_Hidden : BOOL := FALSE;
  Distributed_Safety_Reality_Epoch : UDINT := 0;
END_VAR

{attribute 'qualified_only'}
VAR_GLOBAL  (* GVL_IO_Binding_Runtime *)
  G_Flood_Sensor_Value : ARRAY[1..64] OF BOOL;
  G_Flood_Sensor_Valid : ARRAY[1..64] OF BOOL;
  G_Water_Valve_Open_FB_Value : ARRAY[1..64] OF BOOL;
  G_Water_Valve_Open_FB_Valid : ARRAY[1..64] OF BOOL;
  G_Water_Valve_Close_FB_Value : ARRAY[1..64] OF BOOL;
  G_Water_Valve_Close_FB_Valid : ARRAY[1..64] OF BOOL;
  G_Water_Valve_Output_Channel_Valid : ARRAY[1..64] OF BOOL;
  G_Runtime_Valid : BOOL;
  G_Last_Update_MS : UDINT;
  G_Any_Invalid_Binding : BOOL;
  G_Any_Missing_Binding : BOOL;
  G_Status_Code : UINT;
  G_Status_Text : STRING(128);
END_VAR

VAR_GLOBAL  (* GVL_DISTRIBUTED_COMMIT *)
  Distributed_Commit_Epoch : ULINT := 0;
  Distributed_Commit_Reconciliation_Epoch : ULINT := 0;
  Local_Publication_Commit_Epoch : ULINT := 0;
  Peer_Publication_Commit_Epoch : ULINT := 0;
  Local_Prepare_Epoch : ULINT := 0;
  Peer_Prepare_Epoch : ULINT := 0;
  Publication_Prepare_Active : BOOL := FALSE;
  Publication_Prepare_Valid : BOOL := FALSE;
  Publication_Commit_Requested : BOOL := FALSE;
  Publication_Commit_Confirmed : BOOL := FALSE;
  Peer_Commit_Ack_Valid : BOOL := FALSE;
  Peer_Commit_Ack_Expired : BOOL := FALSE;
  Peer_Commit_Mismatch : BOOL := FALSE;
  Peer_Commit_Replay_Detected : BOOL := FALSE;
  Peer_Commit_Missing : BOOL := FALSE;
  Commit_Lease_Active : BOOL := FALSE;
  Commit_Lease_Expired : BOOL := FALSE;
  Commit_Timeout_MS : UDINT := 5000;
  Local_Commit_Last_Refresh_MS : UDINT := 0;
  Peer_Commit_Last_Refresh_MS : UDINT := 0;
  Commit_Last_Reconciliation_MS : UDINT := 0;
  Distributed_Commit_Valid : BOOL := FALSE;
  Distributed_Commit_Quarantine_Active : BOOL := FALSE;
  Distributed_Commit_Last_Error_Code : UDINT := 0;
  Distributed_Commit_Last_Error_Text : STRING(160) := '';
END_VAR

VAR_GLOBAL  (* GVL_SEMANTIC_EPOCH_INVARIANCE_FABRIC *)
  Semantic_Epoch_Invariance_Valid : BOOL := FALSE;
  Semantic_Epoch_Invariance_Granted : BOOL := FALSE;
  Semantic_Epoch_Invariance_Quarantine_Active : BOOL := TRUE;
  Authority_Semantics_Invariant : BOOL := FALSE;
  CrossEpoch_Permission_Mapping_Stable : BOOL := FALSE;
  Semantic_Intent_Continuity_Valid : BOOL := FALSE;
  Governance_Meaning_Preservation_Coherent : BOOL := FALSE;
  Semantic_Evolution_Lineage_Traceable : BOOL := FALSE;
  Explicit_Semantic_Migration_Governed : BOOL := FALSE;
  CrossEpoch_Semantic_Equivalence_Valid : BOOL := FALSE;
  Distributed_Semantic_Consensus_Stable : BOOL := FALSE;
  Semantic_Interpretation_Integrity_Valid : BOOL := FALSE;
  Semantic_Authority_Drift_Detected : BOOL := FALSE;
  CrossEpoch_Permission_Reinterpretation : BOOL := FALSE;
  Intent_To_Authority_Mismatch_Detected : BOOL := FALSE;
  Governance_Semantic_Fork_Detected : BOOL := FALSE;
  Semantic_Migration_Lineage_Gap_Detected : BOOL := FALSE;
  Distributed_Semantic_Divergence_Detected : BOOL := FALSE;
  Semantic_Epoch_Invariance_Epoch : UDINT := 0;
  Semantic_Epoch_Invariance_Epoch_Coherent : BOOL := FALSE;
  Semantic_Epoch_Invariance_Last_Update_MS : UDINT := 0;
  Semantic_Epoch_Invariance_Lease_Expired : BOOL := TRUE;
  Semantic_Epoch_Invariance_Last_Error_Code : UDINT := 0;
  Semantic_Epoch_Invariance_Last_Error_Text : STRING(160) := '';
  Semantic_Epoch_Invariance_Invalidation_Count : UDINT := 0;
END_VAR

VAR_GLOBAL  (* GVL_SAFETY_RECOVERY *)
  G_Recovery_Phase : E_Recovery_Phase := IDLE;
  G_Recovery_Active : BOOL := FALSE;
  G_Recovery_Requested : BOOL := FALSE;
  G_Recovery_Manual_Confirm : BOOL := FALSE;
  G_Recovery_Start_MS : UDINT := 0;
  G_Recovery_Stable_Since_MS : UDINT := 0;
  G_Recovery_Cooldown_Start_MS : UDINT := 0;
  G_Recovery_Exit_Allowed : BOOL := FALSE;
  G_Recovery_Abort_Reason : INT := 0;  (* 0=none, 1=safety active, 2=confidence low, 3=timeout *)
END_VAR

VAR_GLOBAL  (* GVL_HA_SESSION_REPLICATION *)
  HA_Replication_Enabled : BOOL := FALSE;
  HA_Channel_Healthy : BOOL := FALSE;
  HA_Last_TX_MS : UDINT := 0;
  HA_Last_RX_MS : UDINT := 0;
  HA_Remote_Session_Valid : BOOL := FALSE;
  HA_Remote_Last_Refresh_MS : UDINT := 0;
  HA_Remote_Runtime_Epoch : ULINT := 0;
  HA_Remote_Snapshot_Epoch : ULINT := 0;
  HA_Remote_Boot_Generation : ULINT := 0;
  HA_Remote_Fencing_Token : ULINT := 0;
  HA_Remote_Publication_Allowed : BOOL := FALSE;
  HA_Remote_Runtime_Healthy : BOOL := FALSE;
  HA_Remote_Distributed_Snapshot_Epoch : ULINT := 0;
  HA_Remote_Runtime_Snapshot_Epoch : ULINT := 0;
  HA_Remote_Publication_Epoch : ULINT := 0;
  HA_Remote_Snapshot_Immutable : BOOL := FALSE;
  HA_Remote_Snapshot_Last_Refresh_MS : UDINT := 0;
  HA_Remote_Publication_Commit_Epoch : ULINT := 0;
  HA_Remote_Prepare_Epoch : ULINT := 0;
  HA_Remote_Commit_Ack_Valid : BOOL := FALSE;
  HA_Remote_Commit_Last_Refresh_MS : UDINT := 0;
END_VAR

VAR_GLOBAL  (* GVL_EXECUTION_PROJECTION_INTEGRITY_FABRIC *)
  Execution_Projection_Integrity_Valid : BOOL := FALSE;
  Execution_Projection_Integrity_Granted : BOOL := FALSE;
  Execution_Projection_Integrity_Quarantine_Active : BOOL := TRUE;
  Execution_Authority_Projection_Consistent : BOOL := FALSE;
  CrossDomain_Actuation_Enforcement_Aligned : BOOL := FALSE;
  Physical_Execution_Governance_Canonical : BOOL := FALSE;
  Actuation_Surface_Consensus_Valid : BOOL := FALSE;
  Execution_Projection_Lineage_Coherent : BOOL := FALSE;
  Runtime_Actuation_Projection_Stable : BOOL := FALSE;
  Distributed_Execution_Equivalence_Valid : BOOL := FALSE;
  Execution_Governance_Causality_Grounded : BOOL := FALSE;
  Physical_Enforcement_Timeline_Monotonic : BOOL := FALSE;
  Execution_Projection_Divergence_Detected : BOOL := FALSE;
  Actuation_Path_Authority_Bypass_Detected : BOOL := FALSE;
  CrossDomain_Enforcement_Fork_Detected : BOOL := FALSE;
  Canonical_Governance_Execution_Lost : BOOL := FALSE;
  Runtime_Execution_Lineage_Drift_Detected : BOOL := FALSE;
  Distributed_Actuation_Reality_Fork_Detected : BOOL := FALSE;
  Execution_Projection_Integrity_Epoch : UDINT := 0;
  Execution_Projection_Integrity_Epoch_Coherent : BOOL := FALSE;
  Execution_Projection_Integrity_Last_Update_MS : UDINT := 0;
  Execution_Projection_Integrity_Lease_Expired : BOOL := TRUE;
  Execution_Projection_Integrity_Last_Error_Code : UDINT := 0;
  Execution_Projection_Integrity_Last_Error_Text : STRING(160) := '';
  Execution_Projection_Integrity_Invalidation_Count : UDINT := 0;
END_VAR

{attribute 'qualified_only'}
VAR_GLOBAL  (* GVL_Distributed_Projection_Ownership *)
  G_Projection_Ownership : ARRAY[1..128] OF ST_Distributed_Projection_Ownership;
END_VAR

VAR_GLOBAL  (* GVL_DEGRADED *)
  G_System_Degraded : BOOL := FALSE;
  G_Degraded_Mode_Active : BOOL := FALSE;
  G_Degraded_Recovery_Required : BOOL := FALSE;
END_VAR

{attribute 'qualified_only'}
VAR_GLOBAL  (* GVL_Heating_Runtime_Projection *)
  G_Circuit_Projection : ARRAY[1..GVL_CONSTANTS.C_MAX_HEATING_CIRCUITS] OF ST_Heating_Circuit_Runtime_Projection;
END_VAR

{attribute 'qualified_only'}
VAR_GLOBAL  (* GVL_SYSTEM_SIZE_CONFIG *)
  G_Active_Heating_Circuits : INT := GVL_CONSTANTS.C_MAX_HEATING_CIRCUITS;
  G_Active_Water_Zones : INT := GVL_CONSTANTS.C_MAX_WATER_ZONES;
  G_Active_Light_Zones : INT := GVL_CONSTANTS.C_MAX_LIGHT_ZONES;
  G_Active_Blinds : INT := GVL_CONSTANTS.C_MAX_BLINDS;
  G_Active_Sockets : INT := GVL_CONSTANTS.C_MAX_SOCKETS;
END_VAR

{attribute 'qualified_only'}
VAR_GLOBAL  (* GVL_CONFIG_BACKUP *)
  G_Backup_FloorHeating_Configs : ARRAY[1..GVL_CONSTANTS.C_MAX_HEATING_CIRCUITS] OF ST_FloorHeating_Circuit_Config;
  G_Backup_Max_Active_Manifolds : INT := 0;
  G_Backup_Max_Thermal_Budget : REAL := 0.0;
  G_Backup_Valid : BOOL := FALSE;
END_VAR

{attribute 'qualified_only'}
VAR_GLOBAL  (* GVL_COMMAND_POLICY_CONFIG *)
  G_PLC_Inactive_Close_Gas : BOOL := TRUE;
  G_PLC_Inactive_Stop_Boiler : BOOL := TRUE;
  G_PLC_Inactive_Block_Heating : BOOL := TRUE;
  G_PLC_Inactive_Stop_Vent : BOOL := TRUE;
  G_PLC_Inactive_Block_Water : BOOL := TRUE;
  G_Fire_Block_Heating : BOOL := TRUE;
  G_Fire_Stop_Boiler : BOOL := TRUE;
  G_Fire_Stop_Vent : BOOL := TRUE;
  G_Fire_Open_Lock_1 : BOOL := TRUE;
  G_Fire_Open_Lock_2 : BOOL := TRUE;
  G_Fire_Open_Gate : BOOL := TRUE;
  G_Fire_Open_Wicket : BOOL := TRUE;
  G_Fire_Block_Lock_Close : BOOL := TRUE;
  G_Gas_Close_Gas : BOOL := TRUE;
  G_Gas_Stop_Boiler : BOOL := TRUE;
  G_Gas_Block_Heating : BOOL := TRUE;
  G_Gas_Open_Gate : BOOL := TRUE;
  G_Gas_Open_Wicket : BOOL := TRUE;
  G_Gas_Open_Lock_1 : BOOL := FALSE;
  G_Gas_Open_Lock_2 : BOOL := FALSE;
  G_Water_Block_Water : BOOL := TRUE;
  G_GlobalStop_Block_Heating : BOOL := TRUE;
  G_GlobalStop_Stop_Boiler : BOOL := TRUE;
  G_GlobalStop_Stop_Vent : BOOL := TRUE;
  G_GlobalStop_Block_Water : BOOL := TRUE;
  G_Block_Close_When_Open_Commanded : BOOL := TRUE;
END_VAR

{attribute 'qualified_only'}
VAR_GLOBAL  (* GVL_CONFIG *)
  G_Heating_Config : ST_Heating_Config;
  G_DHW_Config : ST_DHW_Config;
  G_Security_Config : ST_Security_Global_Config;
  G_HMI_FloorHeating_Configs : ARRAY[1..GVL_CONSTANTS.C_MAX_HEATING_CIRCUITS] OF ST_FloorHeating_Circuit_Config;
  G_Heating_Circuit_To_Zone : ARRAY[1..GVL_CONSTANTS.C_MAX_HEATING_CIRCUITS] OF INT := [1, 2, 3, 4, 5, 6, 7, 8, 9, 10, 11, 12, 13, 14, 15, 16];
  G_Wet_Zone_Map : ARRAY[1..32] OF BOOL;
  G_HMI_Tariff_Settings : ST_Tariff_Config;
  G_HMI_Vent_Global_Config : ST_Ventilation_Global_Config;
  G_HMI_Scenario_Configs : ARRAY[1..GVL_CONSTANTS.C_MAX_SCENARIOS] OF ST_Scenario_Config;
  G_HMI_Flood_Config : ST_Flood_Global_Config;
  G_Flood_Global_Config : ST_Flood_Global_Config;
  G_HMI_User_Rules : ARRAY[1..GVL_CONSTANTS.C_MAX_RULES] OF ST_User_Rule;
  G_Calib_Outdoor_Temp : ST_Sensor_Calibration_Record;
  G_Calib_Supply_Temps : ARRAY[1..GVL_CONSTANTS.C_MAX_SUPPLY_TEMPS] OF ST_Sensor_Calibration_Record;
  G_Calib_Room_Temps : ARRAY[1..GVL_CONSTANTS.C_MAX_ZONES] OF ST_Sensor_Calibration_Record;
  G_Calib_Floor_Temps : ARRAY[1..GVL_CONSTANTS.C_MAX_ZONES] OF ST_Sensor_Calibration_Record;
  G_Calib_CO2 : ARRAY[1..GVL_CONSTANTS.C_MAX_ZONES] OF ST_Sensor_Calibration_Record;
  G_Calib_Humidity : ARRAY[1..GVL_CONSTANTS.C_MAX_ZONES] OF ST_Sensor_Calibration_Record;
  G_Calib_Manifold_T_Supply : ARRAY[1..GVL_CONSTANTS.C_MAX_MANIFOLDS] OF ST_Sensor_Calibration_Record;
  G_Calib_Manifold_T_Return : ARRAY[1..GVL_CONSTANTS.C_MAX_MANIFOLDS] OF ST_Sensor_Calibration_Record;
  G_Calib_Methane : ARRAY[1..GVL_CONSTANTS.C_MAX_METHANE_SENSORS] OF ST_Sensor_Calibration_Record;
  G_Calib_CO : ARRAY[1..GVL_CONSTANTS.C_MAX_CO_SENSORS] OF ST_Sensor_Calibration_Record;
  G_Valve_Test_Config : ARRAY[1..GVL_CONSTANTS.C_MAX_MANIFOLDS] OF ST_Valve_Test_Config;
  G_HMI_Apply_Settings : BOOL;
  G_HMI_Mute_Alarm : BOOL;
  G_HMI_Ack_Alarms : BOOL;
  G_HMI_Gate_Open_Req : BOOL;
  G_HMI_Wicket_Open_Req : BOOL;
  G_HMI_Lock_1_Open_Req : BOOL;
  G_HMI_Lock_1_Close_Req : BOOL;
  G_HMI_Lock_2_Open_Req : BOOL;
  G_HMI_Lock_2_Close_Req : BOOL;
  G_Access_Pulse_MS : UDINT := 500;
  G_Allowed_IPs : ARRAY[1..GVL_CONSTANTS.C_MAX_ALLOWED_IPS] OF STRING(15) := ['192.168.1.100', '192.168.1.101', '127.0.0.1', '', ''];
  G_Backup_Circulation_Pump_In_Service : BOOL := TRUE;
  G_Electric_Heater_In_Service : BOOL := TRUE;
  G_Freeze_Hardware_Retry_Count : INT := 2;
  G_Freeze_Hardware_Retry_Delay_MS : UDINT := 5000;
  G_Pump_Exercise_Enabled : BOOL := TRUE;
  G_Pump_Exercise_Interval_MS : UDINT := 604800000;
  G_Pump_Exercise_Duration_MS : UDINT := 30000;
  G_Manifold_Pump_In_Service : ARRAY[1..GVL_CONSTANTS.C_MAX_MANIFOLDS] OF BOOL := [TRUE, TRUE, TRUE, TRUE, TRUE];
  G_Manifold_Priority : ARRAY[1..GVL_CONSTANTS.C_MAX_MANIFOLDS] OF INT := [3, 3, 2, 2, 1];
  G_Manifold_Thermal_Weight : ARRAY[1..GVL_CONSTANTS.C_MAX_MANIFOLDS] OF REAL := [1.0, 1.0, 0.8, 0.8, 0.5];
  G_Max_Active_Manifolds : INT := 3;
  G_Max_Thermal_Budget : REAL := 6.0;
  G_Policy_Min_Hold_MS : UDINT := 300000;
  G_DHW_Heating_Pump_In_Service : BOOL := TRUE;
  G_DHW_Circ_Pump_In_Service : BOOL := TRUE;
  G_Water_Valve_Exercise_Enabled : BOOL := TRUE;
  G_Water_Valve_Exercise_Interval_MS : UDINT := 604800000;
  G_Water_Valve_Exercise_Duration_MS : UDINT := 15000;
  G_Water_Valve_Close_Retry_Count : INT := 2;
  G_Water_Valve_Close_Retry_Delay_MS : UDINT := 3000;
  G_OpenTherm_Enabled : BOOL := FALSE;
  G_OpenTherm_Heartbeat_Timeout_MS : UDINT := 5000;
  G_OpenTherm_Command_Ack_Timeout_MS : UDINT := 3000;
  G_OpenTherm_Register_Map : ARRAY[1..GVL_CONSTANTS.C_MAX_BOILERS] OF ST_OpenTherm_Register_Map;
  G_Modbus_RTU_Driver_Attached : BOOL := FALSE;
  G_Modbus_RTU_Port_Number : BYTE := 1;  (* 1=COM1, 2=COM2, 3=COM3, 4=COM4 *)
  G_Modbus_RTU_Baudrate : UDINT := 9600;
  G_Modbus_RTU_Parity : BYTE := 1;  (* 0=None, 1=Even, 2=Odd *)
  G_Modbus_RTU_Stop_Bits : BYTE := 1;  (* 1 or 2 *)
  G_Modbus_RTU_Data_Bits : BYTE := 8;  (* usually 8 *)
  G_Modbus_RTU_Slave_ID : BYTE := 1;
  G_Modbus_RTU_Poll_Interval_MS : UDINT := 100;
  G_Modbus_RTU_Request_Timeout_MS : UDINT := 250;
  G_Modbus_RTU_Retry_Count : INT := 2;
  G_FloorTemp_Map : ARRAY[1..GVL_CONSTANTS.C_MAX_HEATING_CIRCUITS] OF INT := [1, 2, 3, 4, 5, 6, 7, 8, 9, 10, 11, 12, 13, 14, 15, 16];
  G_RoomTemp_Map : ARRAY[1..16] OF INT := [1, 2, 3, 4, 5, 6, 7, 8, 9, 10, 11, 12, 13, 14, 15, 16];
  G_Door_Map : ARRAY[1..GVL_CONSTANTS.C_MAX_DOOR_SENSORS] OF INT := [1, 2, 3, 4, 5, 6, 7, 8];
  G_Window_Map : ARRAY[1..16] OF INT := [9, 10, 11, 12, 13, 14, 15, 16, 17, 18, 19, 20, 21, 22, 23, 24];
  C_MAX_LIGHT_ZONES : INT := 32;
  G_Evac_Exit_Zones : ARRAY[1..32] OF BOOL;
  G_Evac_Zone_Names : ARRAY[1..32] OF STRING(80);
END_VAR

{attribute 'qualified_only'}
VAR_GLOBAL  (* GVL_HMI_Config_Workflow *)
  G_Open_Editor_Request : BOOL;
  G_Validate_Request : BOOL;
  G_Activate_Request : BOOL;
  G_Rollback_Request : BOOL;
  G_Service_Mode_Active : BOOL;
  G_Operator_Ack : BOOL;
  G_Workflow_State : ST_HMI_Config_Workflow_State;
  G_Runtime_Valid : BOOL;
  G_Last_Update_MS : UDINT;
  G_Status_Code : UINT;
  G_Status_Text : STRING(160);
END_VAR

VAR_GLOBAL  (* GVL_DISTRIBUTED_EPOCH *)
  Distributed_Epoch : ULINT := 0;
  Distributed_Reconciliation_Epoch : ULINT := 0;
  Local_Runtime_Epoch : ULINT := 0;
  Peer_Runtime_Epoch : ULINT := 0;
  Local_Snapshot_Epoch : ULINT := 0;
  Peer_Snapshot_Epoch : ULINT := 0;
  Local_Boot_Generation : ULINT := 0;
  Peer_Boot_Generation : ULINT := 0;
  Local_Fencing_Token : ULINT := 0;
  Peer_Fencing_Token : ULINT := 0;
  Distributed_Epoch_Consistent : BOOL := FALSE;
  Distributed_Reconciliation_Valid : BOOL := FALSE;
  Distributed_Publication_Allowed : BOOL := FALSE;
  Peer_Lease_Active : BOOL := FALSE;
  Peer_Lease_Expired : BOOL := FALSE;
  Peer_Lease_Timeout_MS : UDINT := 5000;
  Peer_Last_Refresh_MS : UDINT := 0;
  Peer_Last_Reconciliation_MS : UDINT := 0;
  Peer_Snapshot_Stale : BOOL := FALSE;
  Peer_Runtime_Stale : BOOL := FALSE;
  Peer_Boot_Mismatch : BOOL := FALSE;
  Peer_Fencing_Conflict : BOOL := FALSE;
  Peer_Semantic_Continuity_Lost : BOOL := FALSE;
  Distributed_Quarantine_Active : BOOL := FALSE;
  Distributed_Last_Error_Code : UDINT := 0;
  Distributed_Last_Error_Text : STRING(160) := '';
END_VAR

{attribute 'qualified_only'}
VAR_GLOBAL  (* GVL_MODE *)
  G_Current_Behavior_Mode : E_Behavior_Mode := BEHAVIOR_HOME;
  G_Mode_Last_Change_TS : UDINT := 0;
  G_Mode_Code : UDINT := 0;
  G_Away_Request : BOOL := FALSE;
  G_Maintenance_Request : BOOL := FALSE;
END_VAR

VAR_GLOBAL  (* GVL_ENVIRONMENTAL_AUTHORITY *)
  Environmental_Authority_Valid : BOOL := FALSE;
  Environmental_Authority_Granted : BOOL := FALSE;
  Environmental_Quarantine_Active : BOOL := TRUE;
  External_Environment_Causally_Compatible : BOOL := FALSE;
  Utility_Environment_Stable : BOOL := FALSE;
  Hydraulic_Source_Stable : BOOL := FALSE;
  Thermal_Environment_Stable : BOOL := FALSE;
  Airflow_Environment_Stable : BOOL := FALSE;
  Mains_Quality_Valid : BOOL := FALSE;
  Supply_Water_Available : BOOL := FALSE;
  Outdoor_Airflow_Valid : BOOL := FALSE;
  Freeze_Protection_Valid : BOOL := FALSE;
  Freeze_Front_Propagation_Detected : BOOL := FALSE;
  Utility_Instability_Propagation_Detected : BOOL := FALSE;
  External_Hydraulic_Collapse_Detected : BOOL := FALSE;
  Airflow_Icing_Condition_Detected : BOOL := FALSE;
  Environmental_Rebound_Race_Detected : BOOL := FALSE;
  Environmental_Authority_Epoch : UDINT := 0;
  Environmental_Authority_Epoch_Coherent : BOOL := FALSE;
  Environmental_Last_Update_MS : UDINT := 0;
  Environmental_Lease_Expired : BOOL := TRUE;
  Environmental_Last_Error_Code : UDINT := 0;
  Environmental_Last_Error_Text : STRING(160) := '';
  Environmental_Invalidation_Count : UDINT := 0;
END_VAR

VAR_GLOBAL  (* GVL_PHYSICAL_AUTHORITY_EPOCH *)
  Physical_Authority_Epoch : UDINT := 0;
  Physical_Authority_Epoch_Valid : BOOL := FALSE;
  Snapshot_Epoch_Coherent : BOOL := FALSE;
  Consensus_Epoch_Coherent : BOOL := FALSE;
  Causality_Epoch_Coherent : BOOL := FALSE;
  PreOutput_Epoch_Coherent : BOOL := FALSE;
  Physical_Epoch_Drift_Detected : BOOL := FALSE;
  Physical_Epoch_Replay_Suspected : BOOL := FALSE;
  Partial_Epoch_Advancement_Detected : BOOL := FALSE;
  Cross_Cycle_Epoch_Skew_Detected : BOOL := FALSE;
  Physical_Authority_Lease_Expired : BOOL := TRUE;
  Physical_Authority_Quarantine_Active : BOOL := TRUE;
  Physical_Authority_Last_Update_MS : UDINT := 0;
  Physical_Authority_Last_Error_Code : UDINT := 0;
  Physical_Authority_Last_Error_Text : STRING(160) := '';
  Physical_Authority_Invalidation_Count : UDINT := 0;
END_VAR

{attribute 'qualified_only'}
VAR_GLOBAL  (* GVL_CONFIG_SIMULATION *)
  G_Simulation_Request : BOOL := FALSE;
  G_Simulation_Confirm : BOOL := FALSE;
  G_Simulation_Result_OK : BOOL := TRUE;
  G_Simulation_Error_Text : STRING(200) := '';
  G_Simulation_Last_Run_MS : UDINT := 0;
END_VAR

VAR_GLOBAL  (* GVL_RUNTIME_EPOCH *)
  Runtime_Epoch : ULINT := 0;
  Runtime_Snapshot_Valid : BOOL := FALSE;
  Runtime_Snapshot_Published : BOOL := FALSE;
  Runtime_Runtime_Barrier_OK : BOOL := TRUE;
  Runtime_Impossible_State_Detected : BOOL := FALSE;
  Runtime_Last_Validation_Time_MS : UDINT := 0;
  Runtime_Last_Error_Code : UDINT := 0;
  Runtime_Last_Error_Text : STRING(160) := '';
  Runtime_Cycle_Start_MS : UDINT := 0;
  Runtime_Cycle_End_MS : UDINT := 0;
  Runtime_PLC_Authority_Valid : BOOL := FALSE;
  Runtime_IO_Publication_Allowed : BOOL := FALSE;
  Runtime_Barrier_Block_Count : UDINT := 0;
END_VAR

{attribute 'qualified_only'}
VAR_GLOBAL RETAIN  (* GVL_Retain *)
  G_Initialized : BOOL := FALSE;  (* Флаг инициализации retain-переменных *)
  G_NVRAM_Data : ARRAY[0..12799] OF BYTE;  (* 100 * 128 = 12800 байт *)
  G_BlackBox_Buffer : ARRAY[0..GVL_CONSTANTS.C_MAX_BLACKBOX_RECORDS-1] OF ST_BlackBox_Record;
  G_BlackBox_LastIndex : INT;
  G_BlackBox_Frozen : BOOL;
  G_Presence_History : ARRAY[0..GVL_CONSTANTS.C_MAX_PRESENCE_HISTORY-1] OF WORD;  (* 168 часов * 6 записей в час = 1008 записей (битовая маска 16 ламп) *)
  G_History_Buffer : ARRAY[1..GVL_CONSTANTS.C_MAX_HISTORY_RECORDS] OF ST_History_Record;
  G_History_Write_Idx : INT := 1;
  G_History_Total_Events : UDINT;
  G_Boiler_Accumulated_MS : ARRAY[1..GVL_CONSTANTS.C_MAX_BOILERS] OF UDINT;
  G_Boiler_Work_Seconds : ARRAY[1..GVL_CONSTANTS.C_MAX_BOILERS] OF UDINT;
  G_Valve_Test_Results : ARRAY[1..GVL_CONSTANTS.C_MAX_MANIFOLDS] OF BOOL;
  G_Access_Codes : ARRAY[1..GVL_CONSTANTS.C_MAX_ACCESS_CODES] OF DWORD := [16#9BE3E0A3, 16#4A89A12D, 16#F4DBDF21, 16#90F59C65, 16#0972D346, 0, 0, 0, 0, 0];
  G_RFID_Tags : ARRAY[1..GVL_CONSTANTS.C_MAX_ACCESS_CODES] OF STRING(20) := ['A1B2C3D4', 'E5F67890', '', '', '', '', '', '', '', ''];
END_VAR

VAR_GLOBAL  (* GVL_SURVIVABILITY_INTELLIGENCE_FABRIC *)
  Survivability_Intelligence_Active : BOOL := TRUE;
  Survivability_Intelligence_ReadOnly : BOOL := TRUE;
  Survivability_Intelligence_NoActuation : BOOL := TRUE;
  Survivability_Intelligence_NoAuthorityMutation : BOOL := TRUE;
  Survivability_Intelligence_NoRecoveryMutation : BOOL := TRUE;
  System_Survivable : BOOL := FALSE;
  Degraded_But_Safe : BOOL := FALSE;
  Isolated_But_Stable : BOOL := FALSE;
  Partitioned_But_Survivable : BOOL := FALSE;
  Resource_Starved_But_Recoverable : BOOL := FALSE;
  Essential_Functions_Preserved : BOOL := FALSE;
  NonEssential_Shedding_Recommended : BOOL := FALSE;
  Telemetry_Rate_Reduction_Recommended : BOOL := FALSE;
  Heavy_Diagnostics_Defer_Recommended : BOOL := FALSE;
  Trend_Analytics_Defer_Recommended : BOOL := FALSE;
  Simulation_Defer_Recommended : BOOL := FALSE;
  LongDuration_Degradation_Observed : BOOL := FALSE;
  Chronic_Degradation_Risk_Increasing : BOOL := FALSE;
  Survivability_Pressure_Observed : BOOL := FALSE;
  Governance_Saturation_Pressure_Observed : BOOL := FALSE;
  Telemetry_Overload_Pressure_Observed : BOOL := FALSE;
  Distributed_Instability_Pressure_Observed : BOOL := FALSE;
  Survivability_Advisory_Available : BOOL := FALSE;
  Survivability_Advisory_Code : STRING(255) := '';
  Survivability_Intelligence_Epoch : UDINT := 0;
END_VAR

VAR_GLOBAL  (* GVL_OBSERVABILITY_TRUTH *)
  Observability_Truth_Valid : BOOL := FALSE;
  Observability_Truth_Granted : BOOL := FALSE;
  Observability_Truth_Quarantine_Active : BOOL := TRUE;
  HMI_Authority_Coherent : BOOL := FALSE;
  Alarm_Authority_Coherent : BOOL := FALSE;
  Trend_Authority_Coherent : BOOL := FALSE;
  Diagnostics_Authority_Coherent : BOOL := FALSE;
  History_Authority_Coherent : BOOL := FALSE;
  HMI_Epoch_Coherent : BOOL := FALSE;
  Alarm_Publication_Coherent : BOOL := FALSE;
  Trend_Causality_Coherent : BOOL := FALSE;
  Diagnostics_Causality_Coherent : BOOL := FALSE;
  Operator_Visibility_Consistent : BOOL := FALSE;
  Stale_HMI_Epoch_Detected : BOOL := FALSE;
  Alarm_Publication_Lag_Detected : BOOL := FALSE;
  Trend_Causality_Skew_Detected : BOOL := FALSE;
  Diagnostic_Truth_Race_Detected : BOOL := FALSE;
  Operator_Visibility_Fragmentation_Detected : BOOL := FALSE;
  Authority_UI_Divergence_Detected : BOOL := FALSE;
  Observability_Truth_Epoch : UDINT := 0;
  Observability_Truth_Epoch_Coherent : BOOL := FALSE;
  Observability_Last_Update_MS : UDINT := 0;
  Observability_Lease_Expired : BOOL := TRUE;
  Observability_Last_Error_Code : UDINT := 0;
  Observability_Last_Error_Text : STRING(160) := '';
  Observability_Invalidation_Count : UDINT := 0;
END_VAR

VAR_GLOBAL  (* GVL_HEATING_DIAGNOSTICS *)
  G_Manifold_Pressure_Fault : ARRAY[1..16] OF BOOL;
  G_Manifold_Current_Fault : ARRAY[1..16] OF BOOL;
  G_Manifold_Return_Temp_Fault : ARRAY[1..16] OF BOOL;
END_VAR

{attribute 'qualified_only'}
VAR_GLOBAL  (* GVL_TEST_PANEL_DEBUG *)
  G_Test_Description : STRING(200);
  G_Test_What_To_Change : STRING(200);
  G_Test_Expected_Text : STRING(200);
  G_Expected_Summary : STRING(200);
  G_Actual_Summary : STRING(200);
  G_Error_Text : STRING(200);
  G_System_State_Line : STRING(200);
  G_Input_Guest_Preheat_Request : BOOL;
  G_Input_Guest_Preheat_Enabled : BOOL;
  G_Input_Guest_Preheat_Boost : INT;
  G_Input_Max_Thermal_Budget : REAL;
  G_Input_Block_Heating : BOOL;
  G_Input_Safety_Stop : BOOL;
END_VAR

VAR_GLOBAL  (* GVL_ACCESS_OUTPUT *)
  DO_Lock_1_Open : BOOL := FALSE;
  DO_Lock_1_Close : BOOL := FALSE;
  DO_Lock_2_Open : BOOL := FALSE;
  DO_Lock_2_Close : BOOL := FALSE;
  DO_Gate_Open : BOOL := FALSE;
  DO_Wicket_Open : BOOL := FALSE;
END_VAR

VAR_GLOBAL  (* GVL_HEATING_REQUEST *)
  G_Freeze_Request : BOOL := FALSE;
  G_Target_Temperature : REAL := 0.0;
  G_Preheat_Request : BOOL := FALSE;
END_VAR

VAR_GLOBAL  (* GVL_COMPLIANCE_FEDERATION_FABRIC *)
  Compliance_Federation_Valid : BOOL := FALSE;
  Compliance_Federation_Granted : BOOL := FALSE;
  Compliance_Federation_Quarantine_Active : BOOL := TRUE;
  Regulatory_Semantics_Coherent : BOOL := FALSE;
  Certification_Boundary_Valid : BOOL := FALSE;
  Regional_Safety_Envelope_Aligned : BOOL := FALSE;
  Governance_Trust_Boundary_Stable : BOOL := FALSE;
  Policy_Compliance_Coherent : BOOL := FALSE;
  CrossJurisdiction_Authority_Aligned : BOOL := FALSE;
  Compliance_Runtime_Projection_Stable : BOOL := FALSE;
  External_Governance_Interpretation_Valid : BOOL := FALSE;
  Certified_Operational_Semantics_Valid : BOOL := FALSE;
  CrossJurisdiction_Semantic_Drift_Detected : BOOL := FALSE;
  Certification_Boundary_Violation_Detected : BOOL := FALSE;
  Policy_Compliance_Divergence_Detected : BOOL := FALSE;
  Regional_Safety_Envelope_Mismatch_Detected : BOOL := FALSE;
  Regulatory_Trust_Corruption_Detected : BOOL := FALSE;
  Governance_Authority_Leakage_Detected : BOOL := FALSE;
  Compliance_Federation_Epoch : UDINT := 0;
  Compliance_Federation_Epoch_Coherent : BOOL := FALSE;
  Compliance_Federation_Last_Update_MS : UDINT := 0;
  Compliance_Federation_Lease_Expired : BOOL := TRUE;
  Compliance_Federation_Last_Error_Code : UDINT := 0;
  Compliance_Federation_Last_Error_Text : STRING(160) := '';
  Compliance_Federation_Invalidation_Count : UDINT := 0;
END_VAR

VAR_GLOBAL  (* GVL_INDUSTRIAL_MAINTAINABILITY_FABRIC *)
  Industrial_Maintainability_Active : BOOL := TRUE;
  Industrial_Maintainability_ReadOnly : BOOL := TRUE;
  Verification_Runtime_Heat_Observed : BOOL := FALSE;
  Diagnostics_Runtime_Heat_Observed : BOOL := FALSE;
  Observability_Runtime_Heat_Observed : BOOL := FALSE;
  Governance_Runtime_Heat_Observed : BOOL := FALSE;
  Unused_Semantic_Pathways_Observed : BOOL := FALSE;
  Inactive_Governance_Chains_Observed : BOOL := FALSE;
  NonContributing_Verification_Layers_Observed : BOOL := FALSE;
  Semantic_Fossilization_Risk : BOOL := FALSE;
  Semantic_Freeze_Boundary_Active : BOOL := TRUE;
  New_Semantic_Layers_Restricted : BOOL := FALSE;
  Survivability_Justification_Required : BOOL := TRUE;
  Merge_Conflict_Risk_Observed : BOOL := FALSE;
  Audit_Complexity_Pressure_Observed : BOOL := FALSE;
  Maintenance_Entropy_Observed : BOOL := FALSE;
  Industrial_Maintainability_Epoch : UDINT := 0;
END_VAR

VAR_GLOBAL  (* GVL_SYSTEM_HEALTH *)
  G_First_Fault_Active : BOOL;
  G_First_Fault_Type : INT;
  G_First_Fault_Source : INT;
  G_System_Severity : E_System_Severity;
  G_Root_Cause : E_System_Root_Cause;
  G_Watchdog_Fault : BOOL;
END_VAR

VAR_GLOBAL  (* GVL_INTENT_BEHAVIOR *)
  I_Request_Night_Mode : BOOL := FALSE;
  I_Request_Away_Mode : BOOL := FALSE;
  I_Request_Comfort_Mode : BOOL := FALSE;
  I_Request_Energy_Save_Mode : BOOL := FALSE;
  I_Request_Preheat : BOOL := FALSE;
  I_Request_Ventilation_Boost : BOOL := FALSE;
  I_Request_Access_Secure_Mode : BOOL := FALSE;
  I_Target_Comfort_Temperature : REAL := 21.0;
  I_Behavior_Priority : INT := 0;
  I_Score_Comfort : INT := 0;
  I_Score_Night : INT := 0;
  I_Score_Energy_Save : INT := 0;
  I_Score_Preheat : INT := 0;
  I_Score_Vent_Boost : INT := 0;
  I_Score_Access_Secure : INT := 0;
  I_Weight_Comfort : REAL := 0.0;
  I_Weight_Night : REAL := 0.0;
  I_Weight_Energy_Save : REAL := 0.0;
  I_Weight_Preheat : REAL := 0.0;
  I_Weight_Vent_Boost : REAL := 0.0;
  I_Weight_Access_Secure : REAL := 0.0;
  I_Best_VentBoost_Zone : INT := 0;
  I_Selected_Scenario_Code : E_System_Reason_Code := REASON_NONE;
  I_Selected_Scenario_Text : STRING(255) := 'No behavior scenario selected';
  I_Reason_Code : E_System_Reason_Code := REASON_NONE;
  I_Reason_Text : STRING(255) := 'No behavior scenario active';
  I_Last_Update_MS : UDINT := 0;
END_VAR

VAR_GLOBAL  (* GVL_INTENT_USER *)
  I_Source_Valid : BOOL := FALSE;
  I_Last_Update_Cycle : UDINT := 0;
  I_Last_Update_MS : UDINT := 0;
  I_Arm_Request : BOOL := FALSE;
  I_Disarm_Request : BOOL := FALSE;
  I_PIN_Code : STRING(8);
  I_RFID_Tag : STRING(32);
  I_2FA_Code_In : STRING(8);
  I_Gate_Open_Request : BOOL := FALSE;
  I_Wicket_Open_Request : BOOL := FALSE;
  I_Lock_1_Open_Request : BOOL := FALSE;
  I_Lock_1_Close_Request : BOOL := FALSE;
  I_Lock_2_Open_Request : BOOL := FALSE;
  I_Lock_2_Close_Request : BOOL := FALSE;
  I_Dangerous_Action_Request : BOOL := FALSE;
  I_Dangerous_Action_Confirm : BOOL := FALSE;
  I_User_Access_Level : INT := 0;
  I_Water_Valve_Test_Open : BOOL := FALSE;
  I_Water_Valve_Test_Close : BOOL := FALSE;
  I_Water_Valve_Test_Confirm : BOOL := FALSE;
  I_Gas_Valve_Test_Open : BOOL := FALSE;
  I_Gas_Valve_Test_Close : BOOL := FALSE;
  I_Gas_Valve_Test_Confirm : BOOL := FALSE;
  I_Water_Selective_Recover : BOOL := FALSE;
  I_Gas_Selective_Recover : BOOL := FALSE;
  I_Scenario_Request : E_SCENARIO_TYPE := E_SCENARIO_TYPE.SCENARIO_NONE;
  I_Lighting_Override_32 : ARRAY[1..GVL_CONSTANTS.C_MAX_LIGHT_ZONES] OF BYTE;
  I_Blinds_Override_32 : ARRAY[1..GVL_CONSTANTS.C_MAX_BLINDS] OF BYTE;
  I_Socket_Override_32 : ARRAY[1..GVL_CONSTANTS.C_MAX_SOCKETS] OF BOOL;
  I_Reset_Errors : BOOL := FALSE;
  I_Set_Temp_Req : BOOL := FALSE;
  I_Target_Zone : INT := 0;
  I_Target_Temperature : REAL := 0.0;
  I_Set_Vent_Req : BOOL := FALSE;
  I_Target_Vent_Speed : REAL := 0.0;
  I_Set_Config_Req : BOOL := FALSE;
  I_Time_Sync_Req : BOOL := FALSE;
  I_New_Time_MS : UDINT := 0;
  I_Set_Adapt_Profile_Req : BOOL := FALSE;
  I_Set_Adapt_Profile_Confirm : BOOL := FALSE;
  I_Adapt_Profile_Value : E_Adapt_Profile := ADAPT_PROFILE_BALANCED;
END_VAR

VAR_GLOBAL  (* GVL_EPISTEMIC_INTEGRITY_FABRIC *)
  Epistemic_Integrity_Valid : BOOL := FALSE;
  Epistemic_Integrity_Granted : BOOL := FALSE;
  Epistemic_Integrity_Quarantine_Active : BOOL := TRUE;
  Physical_Reality_Model_Coherent : BOOL := FALSE;
  Sensor_Truth_Consensus_Valid : BOOL := FALSE;
  Telemetry_Reality_Alignment_Stable : BOOL := FALSE;
  Distributed_Reality_Model_Consistent : BOOL := FALSE;
  Causal_Model_Physically_Valid : BOOL := FALSE;
  Historical_Reality_Anchoring_Valid : BOOL := FALSE;
  Physical_Truth_Lineage_Coherent : BOOL := FALSE;
  Reality_Model_Drift_Bounded : BOOL := FALSE;
  Semantic_To_Physical_Causality_Valid : BOOL := FALSE;
  Physically_False_Consensus_Detected : BOOL := FALSE;
  Telemetry_Corruption_Coherent_Detected : BOOL := FALSE;
  Historical_Reality_Divergence_Detected : BOOL := FALSE;
  Sensor_Trust_Erosion_Detected : BOOL := FALSE;
  Causal_Model_Poisoning_Detected : BOOL := FALSE;
  LongTerm_Epistemic_Drift_Detected : BOOL := FALSE;
  Epistemic_Integrity_Epoch : UDINT := 0;
  Epistemic_Integrity_Epoch_Coherent : BOOL := FALSE;
  Epistemic_Integrity_Last_Update_MS : UDINT := 0;
  Epistemic_Integrity_Lease_Expired : BOOL := TRUE;
  Epistemic_Integrity_Last_Error_Code : UDINT := 0;
  Epistemic_Integrity_Last_Error_Text : STRING(160) := '';
  Epistemic_Integrity_Invalidation_Count : UDINT := 0;
END_VAR

{attribute 'qualified_only'}
VAR_GLOBAL  (* GVL_INTENT_POLICY *)
  G_Preheat_Request : BOOL;
  G_Freeze_Request : BOOL;
  G_Zone_Target_Adjustment : ARRAY[1..GVL_CONSTANTS.C_MAX_ZONES] OF REAL;
END_VAR

VAR_GLOBAL  (* GVL_Distributed_Recovery_Lock *)
  G_Recovery_Lock : ST_Distributed_Recovery_Lock;
  G_Runtime_Valid : BOOL := FALSE;
  G_Last_Update_MS : UDINT := 0;
  G_Recovery_Execution_Blocked : BOOL := TRUE;
  G_Rollback_Execution_Blocked : BOOL := TRUE;
  G_Reopen_Execution_Blocked : BOOL := TRUE;
  G_Status_Code : UINT := 0;
  G_Status_Text : STRING(160) := '';
END_VAR

VAR_GLOBAL  (* GVL_ENERGY_ISOLATION_CAUSALITY_FABRIC *)
  Energy_Isolation_Causality_Valid : BOOL := FALSE;
  Energy_Isolation_Causality_Granted : BOOL := FALSE;
  Physical_Energy_Isolation_Valid : BOOL := FALSE;
  Unsafe_Energy_Propagation_Prevented : BOOL := FALSE;
  CrossDomain_Power_Segmentation_Canonical : BOOL := FALSE;
  Energy_Isolation_Lineage_Coherent : BOOL := FALSE;
  Energy_Causality_Grounded : BOOL := FALSE;
  Distributed_Energy_Isolation_Consensus : BOOL := FALSE;
  Residual_Energy_Leakage_Detected : BOOL := FALSE;
  CrossDomain_Power_Backfeed_Detected : BOOL := FALSE;
  SplitEnergy_Topology_Detected : BOOL := FALSE;
  Unsafe_Energy_Propagation_Detected : BOOL := FALSE;
  Energy_Isolation_Epoch : UDINT := 0;
END_VAR

{attribute 'qualified_only'}
VAR_GLOBAL  (* GVL_Water_Output_Reconciliation *)
  G_Reconciliation_State : ARRAY[1..64] OF ST_Water_Output_Reconciliation_State;
  G_Any_Runtime_Mismatch : BOOL;
  G_Any_Confirmation_Mismatch : BOOL;
  G_Any_Conflict_Detected : BOOL;
  G_Runtime_Valid : BOOL;
  G_Last_Update_MS : UDINT;
  G_Status_Code : UINT;
  G_Status_Text : STRING(128);
END_VAR

VAR_GLOBAL  (* GVL_RESOURCE_STARVATION_BOUNDARY_FABRIC *)
  Resource_Starvation_Boundary_Valid : BOOL := FALSE;
  Resource_Starvation_Boundary_Granted : BOOL := FALSE;
  Resource_Starvation_Bounded : BOOL := FALSE;
  Fair_Execution_Scheduling_Valid : BOOL := FALSE;
  Distributed_Resource_Allocation_Stable : BOOL := FALSE;
  Resource_Causality_Grounded : BOOL := FALSE;
  Starvation_Recovery_Stable : BOOL := FALSE;
  Resource_Starvation_Detected : BOOL := FALSE;
  Scheduler_Starvation_Detected : BOOL := FALSE;
  Distributed_Allocation_Deadlock_Detected : BOOL := FALSE;
  Resource_Starvation_Epoch : UDINT := 0;
END_VAR

{attribute 'qualified_only'}
VAR_GLOBAL  (* GVL_PRESENCE *)
  G_Any_Motion : BOOL := FALSE;
  G_Occupied : BOOL := TRUE;
  G_Auto_Away_Request : BOOL := FALSE;
  G_Last_Motion_TS : UDINT := 0;
  G_Zone_Occupied : ARRAY[1..GVL_CONSTANTS.C_MAX_ZONES] OF BOOL;
  G_Zone_Last_Motion_TS : ARRAY[1..GVL_CONSTANTS.C_MAX_ZONES] OF UDINT;
END_VAR

VAR_GLOBAL  (* GVL_CANONICAL_RUNTIME_FABRIC_REGISTRY *)
  Runtime_Fabric_Registry_Active : BOOL := TRUE;
  Runtime_Fabric_Registry_ReadOnly : BOOL := TRUE;
  Current_Governance_Priority_Tier : E_GOVERNANCE_PRIORITY_TIER := TIER_0_SAFETY;
  Tier0_Safety_Active : BOOL := TRUE;
  Tier1_Authority_Active : BOOL := TRUE;
  Tier2_Physical_Truth_Active : BOOL := TRUE;
  Tier3_Survivability_Active : BOOL := TRUE;
  Tier4_Observability_Active : BOOL := TRUE;
  Tier5_Analytics_Active : BOOL := TRUE;
  Temporal_Integrity_Cluster_Active : BOOL := TRUE;
  Authority_Integrity_Cluster_Active : BOOL := TRUE;
  Physical_Reality_Cluster_Active : BOOL := TRUE;
  Operational_Intelligence_Cluster_Active : BOOL := TRUE;
  Survivability_Cluster_Active : BOOL := TRUE;
  Governance_Scattering_Observed : BOOL := FALSE;
  Semantic_Duplication_Observed : BOOL := FALSE;
  Runtime_Complexity_Pressure_Observed : BOOL := FALSE;
  Governance_Depth_Limit_Reached : BOOL := FALSE;
  Semantic_Recursion_Limit_Reached : BOOL := FALSE;
  Verification_Chaining_Limit_Reached : BOOL := FALSE;
  Observability_Amplification_Limit_Reached : BOOL := FALSE;
  Governance_Runtime_Cost_Observed : BOOL := FALSE;
  Verification_Induced_Instability_Risk : BOOL := FALSE;
  Runtime_Fabric_Registry_Epoch : UDINT := 0;
END_VAR

{attribute 'qualified_only'}
VAR_GLOBAL  (* GVL_SIMULATION *)
  G_Simulation_Enable : BOOL := FALSE;
  G_Test_Scenario_ID : INT := 0;  (* 0=manual flags, 1=safety gas, 2=leak+low pressure, 3=sensor+predictive, 4=dual PLC, 5=full stress *)
  G_Test_Start : BOOL := FALSE;
  G_Test_Stop : BOOL := FALSE;
  G_Test_Scenario_Active : BOOL := FALSE;
  G_Test_Started_MS : UDINT := 0;
  G_Test_Duration_MS : UDINT := 30000;
  G_Test_Expected_Result_Code : INT := 0;  (* 0=none, 1=safety, 2=heating degraded, 3=role conflict, 4=full stress *)
  G_Inject_Heating_Sensor_Fault : BOOL := FALSE;
  G_Inject_IO_Fault : BOOL := FALSE;
  G_Inject_Low_Pressure : BOOL := FALSE;
  G_Inject_Predictive_Pump_Fault : BOOL := FALSE;
  G_Inject_Gas_Alarm : BOOL := FALSE;
  G_Inject_Leak_Alarm : BOOL := FALSE;
  G_Inject_Smoke_Alarm : BOOL := FALSE;
  G_Inject_Dual_PLC_Active : BOOL := FALSE;
  G_Sim_Heating_Sensor_Fault : BOOL := FALSE;
  G_Sim_IO_Fault : BOOL := FALSE;
  G_Sim_Low_Pressure : BOOL := FALSE;
  G_Sim_Predictive_Pump_Fault : BOOL := FALSE;
  G_Sim_Gas_Alarm : BOOL := FALSE;
  G_Sim_Leak_Alarm : BOOL := FALSE;
  G_Sim_Smoke_Alarm : BOOL := FALSE;
  G_Sim_Dual_PLC_Active : BOOL := FALSE;
  G_Test_Running : BOOL := FALSE;
  G_Test_Result_OK : BOOL := FALSE;
  G_Test_Last_Result_Text : STRING(128) := 'No test executed';
END_VAR

VAR_GLOBAL  (* GVL_DEBUG_VIEW *)
  D_Current_Time_MS : UDINT := 0;
  D_Safety_Mode : E_Safety_Mode := NORMAL;
  D_Safety_Active : BOOL := FALSE;
  D_Recovery_Phase : E_Recovery_Phase := IDLE;
  D_Recovery_Active : BOOL := FALSE;
  D_Current_Scenario : STRING(255) := '';
  D_Behavior_Reason : STRING(255) := '';
  D_Score_Night : INT := 0;
  D_Score_Preheat : INT := 0;
  D_Score_VentBoost : INT := 0;
  D_Score_AccessSecure : INT := 0;
  D_Intent_Night : BOOL := FALSE;
  D_Intent_Comfort : BOOL := FALSE;
  D_Intent_VentBoost : BOOL := FALSE;
  D_Intent_AccessSecure : BOOL := FALSE;
  D_Heating_Block : BOOL := FALSE;
  D_Vent_Stop : BOOL := FALSE;
  D_Water_Block : BOOL := FALSE;
  D_Access_Open_Active : BOOL := FALSE;
  D_Global_Reason : STRING(255) := '';
  D_Behavior_Why_Active : STRING(255) := '';
  D_Heating_Why_Blocked : STRING(255) := '';
  D_Vent_Why_Stopped : STRING(255) := '';
  D_Water_Why_Closed : STRING(255) := '';
  D_Access_Why_Opened : STRING(255) := '';
  D_Main_VentBoost_Zone : INT := 0;
  D_Main_VentBoost_Zone_Weight : REAL := 0.0;
  D_Main_VentBoost_Zone_Confidence : REAL := 0.0;
  D_Max_VentBoost_Zone_Weight : REAL := 0.0;
  D_Min_VentBoost_Zone_Weight : REAL := 0.0;
  D_Input_Source_Valid : BOOL := FALSE;
  D_Input_Degraded : BOOL := FALSE;
  D_Sensor_Fault : BOOL := FALSE;
  D_Validation_Failed : BOOL := FALSE;
  D_Anomaly_Detected : BOOL := FALSE;
  D_Validation_Reason : STRING(120) := '';
  D_Anomaly_Reason : STRING(120) := '';
  D_Last_Invalid_Zone : INT := 0;
  D_Min_Zone_Confidence : REAL := 1.0;
  D_Worst_Zone : INT := 0;
  D_Ownership_Violation : BOOL := FALSE;
  D_Adapt_Profile : E_Adapt_Profile := ADAPT_PROFILE_BALANCED;
  D_Adapt_Profile_Text : STRING(32) := 'BALANCED';
  D_Last_Trace_Text : STRING(120) := '';
  D_Last_Trace_Time_MS : UDINT := 0;
  D_Last_Trace_Reason : E_System_Reason_Code := REASON_NONE;
END_VAR

VAR_GLOBAL  (* GVL_RUNTIME_SNAPSHOT *)
  Snapshot_Epoch : ULINT := 0;
  Snapshot_Publication_Epoch : ULINT := 0;
  Snapshot_Frozen : BOOL := FALSE;
  Snapshot_Publication_Allowed : BOOL := FALSE;
  Snapshot_Copy_Valid : BOOL := FALSE;
  Snapshot_Isolation_Valid : BOOL := FALSE;
  Snapshot_Mutation_Detected : BOOL := FALSE;
  Snapshot_Runtime_Authority_Valid : BOOL := FALSE;
  Snapshot_Freeze_Start_MS : UDINT := 0;
  Snapshot_Last_Publication_MS : UDINT := 0;
  Snapshot_Last_Error_Code : UDINT := 0;
  Snapshot_Last_Error_Text : STRING(160) := '';
END_VAR

VAR_GLOBAL  (* GVL_TIME_MONOTONIC *)
  Monotonic_Epoch : ULINT := 0;
  Boot_Generation_ID : ULINT := 0;
  Monotonic_Time_Valid : BOOL := FALSE;
  Monotonic_Time_Initialized : BOOL := FALSE;
  Startup_Quarantine_Active : BOOL := TRUE;
  Startup_Quarantine_Release_Allowed : BOOL := FALSE;
  Startup_Quarantine_Start_MS : UDINT := 0;
  Startup_Quarantine_Timeout_MS : UDINT := 10000;
  Time_Rollback_Detected : BOOL := FALSE;
  Retained_Time_Invalid : BOOL := FALSE;
  Time_Overflow_Detected : BOOL := FALSE;
  Last_Monotonic_Time_MS : UDINT := 0;
  Last_Validated_Time_MS : UDINT := 0;
  Monotonic_Last_Error_Code : UDINT := 0;
  Monotonic_Last_Error_Text : STRING(160) := '';
  Monotonic_Invalidation_Count : UDINT := 0;
END_VAR

VAR_GLOBAL  (* GVL_RUNTIME_STATE_ALGEBRA *)
  Current_Runtime_State : E_SYSTEM_RUNTIME_STATE := SYS_SAFE;
  Previous_Runtime_State : E_SYSTEM_RUNTIME_STATE := SYS_SAFE;
  Runtime_State_Transition_Valid : BOOL := FALSE;
  Runtime_State_Lineage_Coherent : BOOL := FALSE;
  Runtime_State_Monotonic : BOOL := FALSE;
  Runtime_State_ReadOnly_Projection : BOOL := TRUE;
  Runtime_State_NoExecutionMutation : BOOL := TRUE;
  Runtime_State_Transition_Observed : BOOL := FALSE;
  Runtime_State_Drift_Observed : BOOL := FALSE;
  Runtime_State_Epoch : UDINT := 0;
END_VAR

VAR_GLOBAL  (* GVL_Heating_Runtime_Observer *)
  G_Runtime_Observer_Lifecycle_State : E_Runtime_Observer_Lifecycle_State := E_Runtime_Observer_Lifecycle_State.ROS_INACTIVE;
  G_Runtime_Observer_Enable_Request : BOOL := FALSE;
  G_Runtime_Observer_Enable_Authorized : BOOL := FALSE;
  G_Runtime_Observer_Enable_Effective : BOOL := FALSE;
  G_Runtime_Observer_Bootstrap_Mode : BOOL := TRUE;
  G_Runtime_Observer_Passive_Mode : BOOL := TRUE;
  G_Runtime_Observer_ReadOnly_Mode : BOOL := TRUE;
  G_Runtime_Observer_Activation_Validated : BOOL := FALSE;
  G_Runtime_Observer_Sequencing_Validated : BOOL := FALSE;
  G_Runtime_Observer_Publication_Validated : BOOL := FALSE;
  G_Runtime_Observer_Rollback_Validated : BOOL := FALSE;
  G_Runtime_Observer_Governance_Locked : BOOL := TRUE;
  G_Runtime_Observer_Runtime_Authority_Disabled : BOOL := TRUE;
  G_Runtime_Observer_Writable_Exports_Disabled : BOOL := TRUE;
  G_Runtime_Observer_Predictive_Disabled : BOOL := TRUE;
  G_Runtime_Observer_Adaptive_Disabled : BOOL := TRUE;
  G_Runtime_Observer_Replay_Disabled : BOOL := TRUE;
  G_Runtime_Observer_Authorization_Valid : BOOL := FALSE;
  G_Runtime_Observer_Authorization_Status_Code : UINT := 0;
  G_Runtime_Observer_Authorization_Status_Text : STRING(128) := 'Heating runtime observer authorization inactive';
END_VAR

VAR_GLOBAL  (* GVL_OPERATOR_SEMANTIC_ALIGNMENT *)
  Operator_Semantic_Alignment_Valid : BOOL := FALSE;
  Operator_Semantic_Alignment_Granted : BOOL := FALSE;
  Operator_Semantic_Alignment_Quarantine_Active : BOOL := TRUE;
  HMI_Semantic_State_Coherent : BOOL := FALSE;
  Operator_Recovery_Intent_Aligned : BOOL := FALSE;
  Alarm_Semantic_Priority_Coherent : BOOL := FALSE;
  Runtime_Explanation_Coherent : BOOL := FALSE;
  Authority_State_Human_Visible : BOOL := FALSE;
  Human_Interpretation_Coherent : BOOL := FALSE;
  Adaptive_Runtime_Visibility_Valid : BOOL := FALSE;
  Semantic_Explanation_Fresh : BOOL := FALSE;
  Operator_Action_Context_Aligned : BOOL := FALSE;
  HMI_Semantic_Lag_Detected : BOOL := FALSE;
  Operator_Interpretation_Skew_Detected : BOOL := FALSE;
  Alarm_Cognition_Mismatch_Detected : BOOL := FALSE;
  Hidden_Authority_State_Detected : BOOL := FALSE;
  Semantic_Explanation_Divergence_Detected : BOOL := FALSE;
  Human_Recovery_Misunderstanding_Detected : BOOL := FALSE;
  Operator_Alignment_Epoch : UDINT := 0;
  Operator_Alignment_Epoch_Coherent : BOOL := FALSE;
  Operator_Alignment_Last_Update_MS : UDINT := 0;
  Operator_Alignment_Lease_Expired : BOOL := TRUE;
  Operator_Alignment_Last_Error_Code : UDINT := 0;
  Operator_Alignment_Last_Error_Text : STRING(160) := '';
  Operator_Alignment_Invalidation_Count : UDINT := 0;
END_VAR

{attribute 'qualified_only'}
VAR_GLOBAL  (* GVL_Heating_Runtime_Meta *)
  G_Runtime_Meta_Supervision : ST_Heating_Runtime_Meta_Supervision;
  G_Runtime_Meta_Publication_Valid : BOOL := FALSE;
  G_Runtime_Meta_Status_Code : UINT := 0;
  G_Runtime_Meta_Status_Text : STRING(128) := 'Heating runtime meta supervision inactive';
END_VAR

{attribute 'qualified_only'}
VAR_GLOBAL  (* GVL_CONFIG_HISTORY *)
  G_History_Version : ARRAY[1..5] OF UDINT;
  G_History_Time_MS : ARRAY[1..5] OF UDINT;
  G_History_Action : ARRAY[1..5] OF STRING(64);
  G_History_Index : INT := 1;
  G_Last_Changed_By_Level : INT := 0;
  G_Last_Action_Text : STRING(128) := '';
END_VAR

VAR_GLOBAL  (* GVL_EXECUTION_PROGRESS_CAUSALITY_FABRIC *)
  Execution_Progress_Causality_Valid : BOOL := FALSE;
  Execution_Progress_Causality_Granted : BOOL := FALSE;
  Progress_Causality_Grounded : BOOL := FALSE;
  Deterministic_Execution_Continuation_Valid : BOOL := FALSE;
  Progress_Lineage_Coherent : BOOL := FALSE;
  Distributed_Progress_Convergence_Valid : BOOL := FALSE;
  Progress_Timeline_Monotonic : BOOL := FALSE;
  Distributed_Execution_Stall_Detected : BOOL := FALSE;
  Execution_Progress_Divergence_Detected : BOOL := FALSE;
  Recovery_Progress_Oscillation_Detected : BOOL := FALSE;
  Execution_Progress_Epoch : UDINT := 0;
END_VAR

VAR_GLOBAL  (* GVL_CROSSDOMAIN_FAILSAFE_CLOSURE_FABRIC *)
  CrossDomain_FailSafe_Closure_Valid : BOOL := FALSE;
  CrossDomain_FailSafe_Closure_Granted : BOOL := FALSE;
  CrossDomain_FailSafe_Closure_Quarantine_Active : BOOL := TRUE;
  CrossDomain_SafeState_Compatibility_Valid : BOOL := FALSE;
  FailSafe_Topology_Closure_Canonical : BOOL := FALSE;
  MultiDomain_SafeTransition_Stable : BOOL := FALSE;
  SafeState_Recovery_Ordering_Bounded : BOOL := FALSE;
  Physical_Domain_Isolation_Coherent : BOOL := FALSE;
  Thermal_Hydraulic_Compatibility_Valid : BOOL := FALSE;
  Ventilation_Heating_Compatibility_Valid : BOOL := FALSE;
  Access_Evacuation_Compatibility_Valid : BOOL := FALSE;
  Power_Recovery_Sequencing_Valid : BOOL := FALSE;
  Distributed_FailSafe_Consensus_Valid : BOOL := FALSE;
  CrossDomain_FailSafe_Conflict_Detected : BOOL := FALSE;
  Unsafe_Recovery_Topology_Detected : BOOL := FALSE;
  CrossDomain_Recovery_Race_Detected : BOOL := FALSE;
  Distributed_SafeState_Fork_Detected : BOOL := FALSE;
  PowerDomain_Unsafe_Reactivation_Detected : BOOL := FALSE;
  MultiDomain_Recovery_Deadlock_Detected : BOOL := FALSE;
  CrossDomain_FailSafe_Closure_Epoch : UDINT := 0;
  CrossDomain_FailSafe_Closure_Epoch_Coherent : BOOL := FALSE;
  CrossDomain_FailSafe_Closure_Last_Update_MS : UDINT := 0;
  CrossDomain_FailSafe_Closure_Lease_Expired : BOOL := TRUE;
  CrossDomain_FailSafe_Closure_Last_Error_Code : UDINT := 0;
  CrossDomain_FailSafe_Closure_Last_Error_Text : STRING(160) := '';
  CrossDomain_FailSafe_Closure_Invalidation_Count : UDINT := 0;
END_VAR

VAR_GLOBAL  (* GVL_VENT_OUTPUT *)
  AO_Supply_Fans : ARRAY[1..GVL_CONSTANTS.C_MAX_SUPPLY_FANS] OF UINT;
  AO_Exhaust_Fans : ARRAY[1..GVL_CONSTANTS.C_MAX_EXHAUST_FANS] OF UINT;
  DO_Vent_Enable : BOOL := FALSE;
END_VAR

{attribute 'qualified_only'}
VAR_GLOBAL  (* GVL_System_Diagnostics_Publication *)
  G_System_Diagnostics : ST_System_Diagnostics;
  G_System_Diagnostics_Publication_Valid : BOOL := FALSE;
  G_System_Diagnostics_Status_Code : UINT := 0;
  G_System_Diagnostics_Status_Text : STRING(128) := 'System diagnostics publication inactive';
END_VAR

{attribute 'qualified_only'}
VAR_GLOBAL  (* GVL_HMI *)
  G_HMI_Heating_Confidence : REAL := 1.0;
  G_HMI_Heating_Confidence_Percent : INT := 100;
  G_HMI_Heating_Reason_Code : INT := 0;
  G_HMI_Heating_Status_Text : STRING(128) := 'OK';
  G_HMI_Heating_Status_Level : INT := 0;  (* 0=OK, 1=WARN, 2=ALARM *)
  G_HMI_Heating_Cascade_Available : BOOL;
  G_HMI_Heating_Cascade_Degraded : BOOL;
  G_HMI_Heating_Cascade_Partial_Capacity : BOOL;
  G_HMI_Heating_Cascade_No_Flame : BOOL;
  G_HMI_Heating_Cascade_Transport_Degraded : BOOL;
  G_HMI_Heating_Cascade_Ignition_Timeout : BOOL;
  G_HMI_Heating_Cascade_Active_Boilers : UINT;
  G_HMI_Heating_Cascade_Available_Boilers : UINT;
  G_HMI_Boiler_OT_Online : ARRAY[1..GVL_CONSTANTS.C_MAX_BOILERS] OF BOOL;
  G_HMI_Boiler_OT_Command_Ack : ARRAY[1..GVL_CONSTANTS.C_MAX_BOILERS] OF BOOL;
  G_HMI_Boiler_OT_Command_Timeout : ARRAY[1..GVL_CONSTANTS.C_MAX_BOILERS] OF BOOL;
  G_HMI_Boiler_OT_Heartbeat_Timeout : ARRAY[1..GVL_CONSTANTS.C_MAX_BOILERS] OF BOOL;
  G_HMI_Boiler_OT_Adapter_Error : ARRAY[1..GVL_CONSTANTS.C_MAX_BOILERS] OF BOOL;
  G_HMI_Boiler_OT_Heartbeat_Age_MS : ARRAY[1..GVL_CONSTANTS.C_MAX_BOILERS] OF UDINT;
  G_HMI_Boiler_OT_Command_Age_MS : ARRAY[1..GVL_CONSTANTS.C_MAX_BOILERS] OF UDINT;
  G_HMI_Boiler_OT_Adapter_State : ARRAY[1..GVL_CONSTANTS.C_MAX_BOILERS] OF E_OpenTherm_Adapter_State;
  G_HMI_Boiler_OT_Error_State : ARRAY[1..GVL_CONSTANTS.C_MAX_BOILERS] OF E_OpenTherm_Error;
  G_HMI_Heating_Predictive_Pressure_Drop : ARRAY[1..GVL_CONSTANTS.C_MAX_MANIFOLDS] OF BOOL;
  G_HMI_Heating_Predictive_Current_Rise : ARRAY[1..GVL_CONSTANTS.C_MAX_MANIFOLDS] OF BOOL;
END_VAR

{attribute 'qualified_only'}
VAR_GLOBAL  (* GVL_Forensic_Journal *)
  G_Journal : ARRAY[1..256] OF ST_Forensic_Journal_Record;
END_VAR

{attribute 'qualified_only'}
VAR_GLOBAL  (* GVL_SCENARIO_CONFIG *)
  G_Night_Start_Hour : INT := 22;
  G_Night_End_Hour : INT := 6;
  G_Access_Secure_Start_Hour : INT := 23;
  G_Access_Secure_End_Hour : INT := 5;
  G_Comfort_Base_Score : REAL := 10.0;
  G_Night_Base_Score : REAL := 40.0;
  G_Preheat_Base_Score : REAL := 50.0;
  G_VentBoost_Base_Score : REAL := 45.0;
  G_AccessSecure_Base_Score : REAL := 30.0;
  G_VentBoost_Humidity_Threshold : REAL := 65.0;
  G_Night_Activation_Threshold : INT := 30;
  G_Comfort_Activation_Threshold : INT := 40;
  G_VentBoost_Activation_Threshold : INT := 40;
  G_AccessSecure_Activation_Threshold : INT := 25;
  G_Fallback_Adapt_Confidence : REAL := 0.5;
  G_Fallback_Input_Confidence : REAL := 0.5;
END_VAR

VAR_GLOBAL  (* GVL_ENERGY_RESURRECTION_BOUNDARY_FABRIC *)
  Energy_Resurrection_Boundary_Valid : BOOL := FALSE;
  Energy_Resurrection_Boundary_Granted : BOOL := FALSE;
  Energy_Resurrection_Causality_Valid : BOOL := FALSE;
  Energy_Authority_Recovery_Bounded : BOOL := FALSE;
  CrossDomain_Energy_Recovery_Stable : BOOL := FALSE;
  Energy_Resurrection_Ordering_Valid : BOOL := FALSE;
  Distributed_Energy_Recovery_Consensus : BOOL := FALSE;
  Unsafe_Energy_Resurrection_Detected : BOOL := FALSE;
  CrossDomain_Energy_Recovery_Race : BOOL := FALSE;
  Energy_Recovery_Fork_Detected : BOOL := FALSE;
  Energy_Resurrection_Epoch : UDINT := 0;
END_VAR

VAR_GLOBAL  (* GVL_INPUT *)
  IN_Last_Update_MS : UDINT := 0;
  IN_Source_Valid : BOOL := FALSE;
  IN_Room_Temps : ARRAY[1..GVL_CONSTANTS.C_MAX_ZONES] OF REAL;
  IN_Floor_Temps : ARRAY[1..GVL_CONSTANTS.C_MAX_HEATING_CIRCUITS] OF REAL;
  IN_Room_Hum : ARRAY[1..GVL_CONSTANTS.C_MAX_ZONES] OF REAL;
  IN_Room_CO2 : ARRAY[1..GVL_CONSTANTS.C_MAX_ZONES] OF REAL;
  IN_Outdoor_Temp : REAL := 0.0;
  IN_Preheat_Request : BOOL := FALSE;
  IN_Freeze_Request : BOOL := FALSE;
  IN_Water_Sensors : ARRAY[1..GVL_CONSTANTS.C_MAX_FLOOD_SENSORS] OF BOOL;
  IN_Smoke_Sensors : ARRAY[1..GVL_CONSTANTS.C_MAX_SMOKE_SENSORS] OF BOOL;
  IN_Methane_Sensors : ARRAY[1..GVL_CONSTANTS.C_MAX_METHANE_SENSORS] OF REAL;
  IN_CO_Sensors : ARRAY[1..GVL_CONSTANTS.C_MAX_CO_SENSORS] OF REAL;
  IN_Input_Degraded : BOOL := FALSE;
  IN_Sensor_Fault : BOOL := FALSE;
  IN_Validation_Failed : BOOL := FALSE;
  IN_Anomaly_Detected : BOOL := FALSE;
  IN_Validation_Reason : STRING(120) := '';
  IN_Anomaly_Reason : STRING(120) := '';
  IN_Last_Invalid_Zone : INT := 0;
  IN_Room_Temp_Prev : ARRAY[1..GVL_CONSTANTS.C_MAX_ZONES] OF REAL;
  IN_Room_Hum_Prev : ARRAY[1..GVL_CONSTANTS.C_MAX_ZONES] OF REAL;
  IN_Last_Change_MS : ARRAY[1..GVL_CONSTANTS.C_MAX_ZONES] OF UDINT;
  IN_Room_Temp_Confidence : ARRAY[1..GVL_CONSTANTS.C_MAX_ZONES] OF REAL;
  IN_Room_Hum_Confidence : ARRAY[1..GVL_CONSTANTS.C_MAX_ZONES] OF REAL;
  IN_Zone_Confidence : ARRAY[1..GVL_CONSTANTS.C_MAX_ZONES] OF REAL;
  IN_Room_Temp_Reputation : ARRAY[1..GVL_CONSTANTS.C_MAX_ZONES] OF REAL;
  IN_Room_Hum_Reputation : ARRAY[1..GVL_CONSTANTS.C_MAX_ZONES] OF REAL;
  IN_Min_Zone_Confidence : REAL := 1.0;
  IN_Worst_Zone : INT := 0;
END_VAR

{attribute 'qualified_only'}
VAR_GLOBAL  (* GVL_Water_Orchestration *)
  G_Traversal_State : ARRAY[1..64] OF ST_Water_Graph_Traversal_State;
  G_Orchestration_State : ARRAY[1..64] OF ST_Water_Orchestration_Runtime_State;
  G_Topology_Version : UDINT;
  G_Config_Runtime_Ready : BOOL;
  G_Any_Traversal_Conflict : BOOL;
  G_Any_Escalation_Required : BOOL;
  G_Runtime_Valid : BOOL;
  G_Last_Update_MS : UDINT;
  G_Status_Code : UINT;
  G_Status_Text : STRING(128);
END_VAR

{attribute 'qualified_only'}
VAR_GLOBAL  (* GVL_Water_Topology_Config *)
  G_Config_Record : ARRAY[1..64] OF ST_Water_Topology_Config_Record;
  G_Active_Config_Version : UDINT;
  G_Config_Loaded : BOOL;
  G_Runtime_Remap_Ready : BOOL;
  G_Any_Invalid_Config : BOOL;
  G_Any_Multi_Valve_Required : BOOL;
  G_Runtime_Valid : BOOL;
  G_Last_Update_MS : UDINT;
  G_Status_Code : UINT;
  G_Status_Text : STRING(128);
END_VAR

VAR_GLOBAL  (* GVL_SAFETY_OBSERVABILITY_TRUTH_FABRIC *)
  Safety_Observability_Truth_Valid : BOOL := FALSE;
  Safety_Observability_Truth_Granted : BOOL := FALSE;
  Safety_Reality_Projection_Valid : BOOL := FALSE;
  Observability_Reality_Equivalence_Granted : BOOL := FALSE;
  Safety_Projection_Causality_Grounded : BOOL := FALSE;
  Physical_Safety_Projection_Canonical : BOOL := FALSE;
  Distributed_Safety_Projection_Consensus : BOOL := FALSE;
  Safety_Observability_Lineage_Coherent : BOOL := FALSE;
  FakeSafe_Projection_Detected : BOOL := FALSE;
  Telemetry_Reality_Divergence_Detected : BOOL := FALSE;
  Stale_Safety_Projection_Detected : BOOL := FALSE;
  Safety_Observability_Fork_Detected : BOOL := FALSE;
  Safety_Observability_Epoch : UDINT := 0;
END_VAR

{attribute 'qualified_only'}
VAR_GLOBAL  (* GVL_Config_Versioning *)
  G_Config_Current_Version : UDINT := 1;
  G_Config_Last_Good_Version : UDINT := 1;
  G_Config_Current_Checksum : UDINT := 0;
  G_Config_Last_Good_Checksum : UDINT := 0;
  G_Config_Rollback_Requested : BOOL := FALSE;
  G_Config_Rollback_Active : BOOL := FALSE;
  G_Config_Invalid_Detected : BOOL := FALSE;
END_VAR

{attribute 'qualified_only'}
VAR_GLOBAL  (* GVL_MODBUS_RTU_BRIDGE *)
  G_Bridge_Enabled : BOOL := FALSE;
  G_Driver_Online : BOOL := FALSE;
  G_Driver_Error : BOOL := FALSE;
  G_Driver_Error_Code : WORD := 0;
  G_Request_Valid : BOOL := FALSE;
  G_Request_Index : INT := 0;
  G_Request_Slave_ID : BYTE := 0;
  G_Request_Function_Code : E_Modbus_Function := MB_NONE;
  G_Request_Start_Register : UINT := 0;
  G_Request_Register_Count : UINT := 0;
  G_Request_Write_Value : ARRAY[1..32] OF WORD;
  G_Request_Sequence : UDINT := 0;
  G_Request_Timeout_MS : UDINT := 0;
  G_Response_Busy : BOOL := FALSE;
  G_Response_Done : BOOL := FALSE;
  G_Response_Error : BOOL := FALSE;
  G_Response_Error_Code : WORD := 0;
  G_Response_Value : ARRAY[1..32] OF WORD;
  G_Response_Sequence : UDINT := 0;
  G_Response_Update_MS : UDINT := 0;
END_VAR

{attribute 'qualified_only'}
VAR_GLOBAL  (* GVL_Water_Recovery_Runtime *)
  G_Recovery_State : ARRAY[1..64] OF ST_Water_Recovery_Runtime_State;
  G_Any_Recovery_Denied : BOOL;
  G_Any_Unsafe_Recovery : BOOL;
  G_Runtime_Valid : BOOL;
  G_Last_Update_MS : UDINT;
  G_Status_Code : UINT;
  G_Status_Text : STRING(128);
END_VAR

VAR_GLOBAL  (* GVL_GOVERNANCE_OBSERVER_CONSENSUS_FABRIC *)
  Governance_Observer_Consensus_Valid : BOOL := FALSE;
  Governance_Observer_Consensus_Granted : BOOL := FALSE;
  Governance_Observer_Consensus_Quarantine_Active : BOOL := TRUE;
  Distributed_Governance_Projection_Consistent : BOOL := FALSE;
  Observer_Semantic_Consensus_Valid : BOOL := FALSE;
  CrossNode_Authority_Interpretation_Aligned : BOOL := FALSE;
  Governance_Reality_Canonical : BOOL := FALSE;
  Observer_Projection_Lineage_Coherent : BOOL := FALSE;
  Canonical_Projection_Vector_Stable : BOOL := FALSE;
  Distributed_Interpretation_Equivalence_Valid : BOOL := FALSE;
  Governance_Projection_Causality_Grounded : BOOL := FALSE;
  Observer_Timeline_Consensus_Monotonic : BOOL := FALSE;
  Observer_Governance_Divergence_Detected : BOOL := FALSE;
  CrossNode_Authority_Interpretation_Fork : BOOL := FALSE;
  Semantic_Projection_Mismatch_Detected : BOOL := FALSE;
  Canonical_Governance_Reality_Lost : BOOL := FALSE;
  Observer_Projection_Lineage_Drift_Detected : BOOL := FALSE;
  Distributed_Governance_Reality_Fork_Detected : BOOL := FALSE;
  Governance_Observer_Consensus_Epoch : UDINT := 0;
  Governance_Observer_Consensus_Epoch_Coherent : BOOL := FALSE;
  Governance_Observer_Consensus_Last_Update_MS : UDINT := 0;
  Governance_Observer_Consensus_Lease_Expired : BOOL := TRUE;
  Governance_Observer_Consensus_Last_Error_Code : UDINT := 0;
  Governance_Observer_Consensus_Last_Error_Text : STRING(160) := '';
  Governance_Observer_Consensus_Invalidation_Count : UDINT := 0;
END_VAR

VAR_GLOBAL  (* GVL_HEATING_OUTPUT *)
  DO_Zone_Valves : ARRAY[1..GVL_CONSTANTS.C_MAX_HEATING_CIRCUITS] OF BOOL;
  DO_Manifold_Pumps : ARRAY[1..GVL_CONSTANTS.C_MAX_MANIFOLDS] OF BOOL;
  AO_Manifold_Valves : ARRAY[1..GVL_CONSTANTS.C_MAX_MANIFOLDS] OF UINT;
  DO_DHW_Heating_Pump : BOOL := FALSE;
  DO_DHW_Circ_Pump : BOOL := FALSE;
  DO_Backup_Circulation_Pump : BOOL := FALSE;
  DO_Electric_Heater_Enable : BOOL := FALSE;
END_VAR

{attribute 'qualified_only'}
VAR_GLOBAL  (* GVL_Heating_Runtime_Supervisory_Publication *)
  G_Publication : ST_Heating_Runtime_Supervisory_Publication;
END_VAR

{attribute 'qualified_only'}
VAR_GLOBAL  (* GVL_Distributed_Execution_Gates *)
  G_Can_Replicate : BOOL;
  G_Can_Execute : BOOL;
  G_Can_Orchestrate : BOOL;
  G_Can_Recover : BOOL;
  G_Can_Rollback : BOOL;
  G_Can_Own_Projection : BOOL;
  G_Runtime_Valid : BOOL;
  G_Last_Update_MS : UDINT;
  G_Status_Code : UINT;
  G_Status_Text : STRING(160);
END_VAR

VAR_GLOBAL  (* GVL_DISTRIBUTED_SNAPSHOT *)
  Distributed_Snapshot_Epoch : ULINT := 0;
  Distributed_Snapshot_Reconciliation_Epoch : ULINT := 0;
  Local_Distributed_Snapshot_Epoch : ULINT := 0;
  Peer_Distributed_Snapshot_Epoch : ULINT := 0;
  Local_Runtime_Snapshot_Epoch : ULINT := 0;
  Peer_Runtime_Snapshot_Epoch : ULINT := 0;
  Local_Publication_Epoch : ULINT := 0;
  Peer_Publication_Epoch : ULINT := 0;
  Distributed_Snapshot_Frozen : BOOL := FALSE;
  Peer_Snapshot_Immutable : BOOL := FALSE;
  Distributed_Publication_Reconciled : BOOL := FALSE;
  Distributed_Publication_Freeze_Valid : BOOL := FALSE;
  Distributed_Snapshot_Consistent : BOOL := FALSE;
  Peer_Publication_Stale : BOOL := FALSE;
  Peer_Snapshot_Not_Immutable : BOOL := FALSE;
  Peer_Publication_Divergence : BOOL := FALSE;
  Peer_Publication_Reconciliation_Lost : BOOL := FALSE;
  Distributed_Snapshot_Quarantine_Active : BOOL := FALSE;
  Peer_Snapshot_Last_Refresh_MS : UDINT := 0;
  Peer_Snapshot_Lease_Active : BOOL := FALSE;
  Peer_Snapshot_Lease_Expired : BOOL := FALSE;
  Peer_Snapshot_Lease_Timeout_MS : UDINT := 5000;
  Distributed_Snapshot_Last_Error_Code : UDINT := 0;
  Distributed_Snapshot_Last_Error_Text : STRING(160) := '';
END_VAR

VAR_GLOBAL  (* GVL_PHYSICAL_SAFESTATE_LATTICE_FABRIC *)
  Physical_SafeState_Lattice_Valid : BOOL := FALSE;
  Physical_SafeState_Lattice_Granted : BOOL := FALSE;
  Physical_SafeState_Lattice_Quarantine_Active : BOOL := TRUE;
  Canonical_SafeState_Topology_Valid : BOOL := FALSE;
  Physical_SafeState_Lattice_Coherent : BOOL := FALSE;
  Deterministic_FailSafe_Convergence_Granted : BOOL := FALSE;
  SafeState_Energy_Boundary_Stable : BOOL := FALSE;
  SafeState_Physical_Risk_Bounded : BOOL := FALSE;
  Heating_SafeState_Compatible : BOOL := FALSE;
  Water_SafeState_Compatible : BOOL := FALSE;
  Ventilation_SafeState_Compatible : BOOL := FALSE;
  Access_SafeState_Compatible : BOOL := FALSE;
  Lighting_SafeState_Compatible : BOOL := FALSE;
  Thermal_SafeState_Stable : BOOL := FALSE;
  Hydraulic_SafeState_Stable : BOOL := FALSE;
  Airflow_SafeState_Stable : BOOL := FALSE;
  Occupancy_SafeState_Stable : BOOL := FALSE;
  Residual_Actuation_Safe : BOOL := FALSE;
  SafeState_Ambiguity_Detected : BOOL := FALSE;
  Partial_SafeState_Asymmetry_Detected : BOOL := FALSE;
  Physical_SafeState_Deadlock_Detected : BOOL := FALSE;
  Unsafe_SafeState_Topology_Detected : BOOL := FALSE;
  Residual_Unsafe_Actuation_Detected : BOOL := FALSE;
  SafeState_Energy_Leakage_Detected : BOOL := FALSE;
  Physical_SafeState_Lattice_Epoch : UDINT := 0;
  Physical_SafeState_Lattice_Epoch_Coherent : BOOL := FALSE;
  Physical_SafeState_Lattice_Last_Update_MS : UDINT := 0;
  Physical_SafeState_Lattice_Lease_Expired : BOOL := TRUE;
  Physical_SafeState_Lattice_Last_Error_Code : UDINT := 0;
  Physical_SafeState_Lattice_Last_Error_Text : STRING(160) := '';
  Physical_SafeState_Lattice_Invalidation_Count : UDINT := 0;
END_VAR

{attribute 'qualified_only'}
VAR_GLOBAL  (* GVL_CONFIG_VALIDATION *)
  G_Config_Valid : BOOL := TRUE;
  G_Config_Critical_Error : BOOL := FALSE;
  G_Config_Force_Safe_Mode : BOOL := TRUE;
  G_Config_Auto_Corrected : BOOL := FALSE;
  G_Config_Reset_To_Default_Done : BOOL := FALSE;
  G_Config_Last_Error_Text : STRING(200) := '';
  G_Config_Last_Action_Text : STRING(200) := '';
  G_Config_Last_Update_MS : UDINT := 0;
END_VAR

VAR_GLOBAL  (* GVL_TRACE *)
  G_Trace_Buffer : ARRAY[1..200] OF ST_Trace_Entry;
  G_Trace_Write_Index : INT := 1;
  G_Trace_Enabled : BOOL := TRUE;
END_VAR

{attribute 'qualified_only'}
VAR_GLOBAL  (* GVL_Water_Topology_Config_Source *)
  G_Source_Record : ARRAY[1..64] OF ST_Water_Topology_Config_Record;
END_VAR

{attribute 'qualified_only'}
VAR_GLOBAL  (* GVL_CONFIG_CONTROL *)
  G_Apply_Request : BOOL := FALSE;
  G_Apply_Confirm : BOOL := FALSE;
  G_Rollback_Request : BOOL := FALSE;
  G_Rollback_Confirm : BOOL := FALSE;
  G_Reset_Default_Request : BOOL := FALSE;
  G_Reset_Default_Confirm : BOOL := FALSE;
  G_Config_Version : UDINT := 1;
  G_Last_Good_Version : UDINT := 1;
  G_Backup_Valid : BOOL := FALSE;
  G_Apply_Done : BOOL := FALSE;
  G_Rollback_Done : BOOL := FALSE;
  STG_Reputation_Learning_Rate : REAL := 0.05;
  STG_Reputation_Recovery_Decay : REAL := 0.01;
  STG_Min_Sensor_Confidence : REAL := 0.1;
  STG_Bad_Spike_Confidence : REAL := 0.3;
  STG_Default_Confidence : REAL := 1.0;
  STG_Night_Start_Hour : INT := 22;
  STG_Night_End_Hour : INT := 6;
  STG_VentBoost_Humidity_Threshold : REAL := 65.0;
  STG_Stabilization_Delay_MS : UDINT := 5000;
  STG_PLC_Inactive_Close_Gas : BOOL := TRUE;
  STG_PLC_Inactive_Stop_Boiler : BOOL := TRUE;
  STG_PLC_Inactive_Block_Heating : BOOL := TRUE;
  STG_PLC_Inactive_Stop_Vent : BOOL := TRUE;
  STG_PLC_Inactive_Block_Water : BOOL := TRUE;
  BCK_Reputation_Learning_Rate : REAL := 0.05;
  BCK_Reputation_Recovery_Decay : REAL := 0.01;
  BCK_Min_Sensor_Confidence : REAL := 0.1;
  BCK_Bad_Spike_Confidence : REAL := 0.3;
  BCK_Default_Confidence : REAL := 1.0;
  BCK_Night_Start_Hour : INT := 22;
  BCK_Night_End_Hour : INT := 6;
  BCK_VentBoost_Humidity_Threshold : REAL := 65.0;
  BCK_Stabilization_Delay_MS : UDINT := 5000;
  BCK_PLC_Inactive_Close_Gas : BOOL := TRUE;
  BCK_PLC_Inactive_Stop_Boiler : BOOL := TRUE;
  BCK_PLC_Inactive_Block_Heating : BOOL := TRUE;
  BCK_PLC_Inactive_Stop_Vent : BOOL := TRUE;
  BCK_PLC_Inactive_Block_Water : BOOL := TRUE;
END_VAR

VAR_GLOBAL  (* GVL_SEMANTIC_COMMIT *)
  Semantic_Commit_Epoch : ULINT := 0;
  Semantic_Checkpoint_Epoch : ULINT := 0;
  Semantic_Publication_Commit_Epoch : ULINT := 0;
  Local_Semantic_Checkpoint_Epoch : ULINT := 0;
  Peer_Semantic_Checkpoint_Epoch : ULINT := 0;
  Local_Semantic_Commit_Epoch : ULINT := 0;
  Peer_Semantic_Commit_Epoch : ULINT := 0;
  Semantic_Checkpoint_Prepare_Active : BOOL := FALSE;
  Semantic_Checkpoint_Prepare_Valid : BOOL := FALSE;
  Semantic_Checkpoint_Ack_Valid : BOOL := FALSE;
  Semantic_Publication_Commit_Requested : BOOL := FALSE;
  Semantic_Publication_Commit_Confirmed : BOOL := FALSE;
  Semantic_Checkpoint_Mismatch : BOOL := FALSE;
  Semantic_Commit_Mismatch : BOOL := FALSE;
  Semantic_Rollback_Detected : BOOL := FALSE;
  Semantic_Replay_Fenced : BOOL := FALSE;
  Semantic_Checkpoint_Missing : BOOL := FALSE;
  Semantic_Checkpoint_Drift_Suspected : BOOL := FALSE;
  Semantic_Checkpoint_Jitter_Suspected : BOOL := FALSE;
  Semantic_Commit_Replay_Storm_Suspected : BOOL := FALSE;
  Semantic_Commit_Stabilization_Required : BOOL := FALSE;
  Semantic_Commit_Stabilized : BOOL := FALSE;
  Semantic_Commit_Stabilization_Window_MS : UDINT := 3000;
  Semantic_Commit_Last_Stable_MS : UDINT := 0;
  Semantic_Drift_Event_Count : ULINT := 0;
  Semantic_Jitter_Event_Count : ULINT := 0;
  Semantic_Replay_Storm_Event_Count : ULINT := 0;
  Semantic_Last_Drift_MS : UDINT := 0;
  Semantic_Last_Jitter_MS : UDINT := 0;
  Semantic_Last_Replay_Storm_MS : UDINT := 0;
  Semantic_Stabilization_Telemetry_Valid : BOOL := FALSE;
  Semantic_Commit_Lease_Active : BOOL := FALSE;
  Semantic_Commit_Lease_Expired : BOOL := FALSE;
  Semantic_Commit_Timeout_MS : UDINT := 5000;
  Semantic_Commit_Last_Refresh_MS : UDINT := 0;
  Peer_Semantic_Commit_Last_Refresh_MS : UDINT := 0;
  Semantic_Commit_Valid : BOOL := FALSE;
  Semantic_Commit_Quarantine_Active : BOOL := FALSE;
  Semantic_Commit_Forced_Safe_Mode : BOOL := FALSE;
  Semantic_Commit_Last_Error_Code : UDINT := 0;
  Semantic_Commit_Last_Error_Text : STRING(160) := '';
  Semantic_Commit_Invalidation_Count : UDINT := 0;
END_VAR

VAR_GLOBAL  (* GVL_COMMAND_SHADOW *)
  G_Gas_Valve_Close : BOOL := FALSE;
  G_Boiler_Stop : BOOL := FALSE;
  G_Supply_100_Req : BOOL := FALSE;
  G_Supply_80_Req : BOOL := FALSE;
  G_Vent_PV3_Boost : BOOL := FALSE;
  G_Exhaust_100_Req : BOOL := FALSE;
  G_Vent_Stop : BOOL := FALSE;
  G_Vent_Block : BOOL := FALSE;
  G_Vent_Smoke_Exhaust : BOOL := FALSE;
  G_Heating_Block : BOOL := FALSE;
  G_Heating_Emergency_Stop : BOOL := FALSE;
  G_Heating_Gas_Safety_Stop : BOOL := FALSE;
  G_Water_Block : BOOL := FALSE;
  G_Water_Emergency_Stop : BOOL := FALSE;
  G_Close_Valve_35 : BOOL := FALSE;
  G_Close_Valve_36 : BOOL := FALSE;
  G_Lock_1_Open : BOOL := FALSE;
  G_Lock_1_Close : BOOL := FALSE;
  G_Lock_2_Open : BOOL := FALSE;
  G_Lock_2_Close : BOOL := FALSE;
  G_Gate_Open : BOOL := FALSE;
  G_Wicket_Open : BOOL := FALSE;
END_VAR

VAR_GLOBAL  (* GVL_PHYSICAL_SAFETY_PROJECTION_FABRIC *)
  Physical_Safety_Projection_Valid : BOOL := FALSE;
  Physical_Safety_Projection_Granted : BOOL := FALSE;
  Physical_Plant_Safety_Projection_Stable : BOOL := FALSE;
  Energy_State_Safety_Projection_Valid : BOOL := FALSE;
  Recovery_State_Safety_Projection_Valid : BOOL := FALSE;
  Physical_Projection_Causality_Valid : BOOL := FALSE;
  Projection_Reality_Alignment_Stable : BOOL := FALSE;
  Physical_Safety_Projection_Drift_Detected : BOOL := FALSE;
  Hidden_Unsafe_Physical_State_Detected : BOOL := FALSE;
  Unsafe_Projection_Backfill_Detected : BOOL := FALSE;
  Physical_Safety_Projection_Epoch : UDINT := 0;
END_VAR

VAR_GLOBAL  (* GVL_GOVERNANCE_VALIDATOR_INTEGRITY_FABRIC *)
  Governance_Validator_Integrity_Valid : BOOL := FALSE;
  Governance_Validator_Integrity_Granted : BOOL := FALSE;
  Governance_Validator_Integrity_Quarantine_Active : BOOL := TRUE;
  Validator_Semantics_Immutable : BOOL := FALSE;
  CrossEpoch_Validation_Equivalence_Stable : BOOL := FALSE;
  Distributed_Validator_Consensus_Valid : BOOL := FALSE;
  Governance_Rule_Integrity_Canonical : BOOL := FALSE;
  Validator_Lineage_Coherent : BOOL := FALSE;
  Validator_Causality_Grounded : BOOL := FALSE;
  Governance_Rule_Evolution_Governed : BOOL := FALSE;
  Distributed_Validation_Timeline_Monotonic : BOOL := FALSE;
  Validator_Interpretation_Equivalence_Valid : BOOL := FALSE;
  Validator_Semantic_Drift_Detected : BOOL := FALSE;
  CrossNode_Validation_Fork : BOOL := FALSE;
  Governance_Rule_Mutation_Detected : BOOL := FALSE;
  SelfReferential_Validator_Corruption : BOOL := FALSE;
  Validator_Lineage_Drift_Detected : BOOL := FALSE;
  Distributed_Validator_Reality_Fork_Detected : BOOL := FALSE;
  Governance_Validator_Integrity_Epoch : UDINT := 0;
  Governance_Validator_Integrity_Epoch_Coherent : BOOL := FALSE;
  Governance_Validator_Integrity_Last_Update_MS : UDINT := 0;
  Governance_Validator_Integrity_Lease_Expired : BOOL := TRUE;
  Governance_Validator_Integrity_Last_Error_Code : UDINT := 0;
  Governance_Validator_Integrity_Last_Error_Text : STRING(160) := '';
  Governance_Validator_Integrity_Invalidation_Count : UDINT := 0;
END_VAR

